KUKA KRL data list: NEW_MASTER_MESA_A.dat

&ACCESS RVP
&REL 381
&PARAM EDITMASK = *
&PARAM TEMPLATE = C:\KRC\Roboter\Template\vorgabe
&PARAM DISKPATH = KRC:\R1\Program\Solda\MASTER_125
DEFDAT  NEW_MASTER_MESA_A
;FOLD EXTERNAL DECLARATIONS;%{PE}%MKUKATPBASIS,%CEXT,%VCOMMON,%P
;FOLD BASISTECH EXT;%{PE}%MKUKATPBASIS,%CEXT,%VEXT,%P
EXT  BAS (BAS_COMMAND  :IN,REAL  :IN )
DECL INT SUCCESS
;ENDFOLD (BASISTECH EXT)
;FOLD USER EXT;%{E}%MKUKATPUSER,%CEXT,%VEXT,%P
;Make your modifications here

;ENDFOLD (USER EXT)
;ENDFOLD (EXTERNAL DECLARATIONS)
DECL ATBg_Start_T AS_WDAT1={JobModeId 1306102413,ParamSetId -1047099609,StartTime 0.0,PreFlowTime 0.0,Channel1 0.0,Channel2 2.00000,Channel3 0.0,Channel4 0.0,Channel5 0.0,Channel6 0.0,Channel7 0.0,Channel8 0.0,PurgeTime 0.0}
DECL ATBg_Weld_T AW_WDAT1={JobModeId -187662529,ParamSetId -430485013,Velocity 0.00830000,Channel1 30.0000,Channel2 1.00000,Channel3 0.0,Channel4 0.0,Channel5 0.0,Channel6 0.0,Channel7 0.0,Channel8 0.0}
DECL WTCg_WeaveDefinition_T WV_WDAT1={Pattern #None,Length 4.00000,Amplitude 2.00000,Angle 0.0}
DECL FDAT FP1={TOOL_NO 1,BASE_NO 0,IPO_FRAME #BASE,POINT2[] " ",TQ_STATE FALSE}
DECL PDAT PPDAT1={ACC 100.000,APO_DIST 100.000,APO_MODE #CPTP,GEAR_JERK 50.0000}
DECL E6POS XP1={X 1496.76196,Y 582.870911,Z 1275.91040,A 159.098511,B 49.1786919,C -124.034058,S 0,T 43,E1 180.001038,E2 179.999084,E3 180.004181,E4 0.0,E5 0.0,E6 0.0}
DECL MODULEPARAM_T LAST_TP_PARAMS={PARAMS[] "Kuka.MoveDataPtpName=PDAT60; Kuka.VelocityPtp=100; Kuka.PointName=P78; Kuka.BlendingEnabled=False; Kuka.FrameData.tq_state=False; Kuka.FrameData.base_no=0; Kuka.FrameData.tool_no=1; Kuka.FrameData.ipo_frame=#BASE; Kuka.MovementDataPdat.apo_mode=#CPTP; Kuka.MovementDataPdat.apo_dist=100; Kuka.MovementData.acc=100; Kuka.MovementData.gear_jerk=50; ArcTech.WdatVarName=WDAT39; Kuka.MoveDataName=CPDAT51; Kuka.VelocityPath=0.3; Kuka.MovementData.apo_fac=50; Kuka.MovementData.apo_dist=100; Kuka.MovementData.axis_acc=100; Kuka.MovementData.axis_vel=100; Kuka.MovementData.circ_typ=#BASE; Kuka.MovementData.exax_ign=0; Kuka.MovementData.jerk_fac=50; Kuka.MovementData.ori_typ=#VAR; Kuka.FrameData.point2=                                                                                                                                                                                                "}
DECL ATBg_Crater_T AC_WDAT2={JobModeId -187662529,ParamSetId -1375177600,CraterTime 0.100000,PostflowTime 0.100000,Channel1 30.0000,Channel2 1.00000,Channel3 0.0,Channel4 0.0,Channel5 0.0,Channel6 0.0,Channel7 0.0,Channel8 0.0,BurnBackTime 0.0}
DECL FDAT FP2={TOOL_NO 1,BASE_NO 0,IPO_FRAME #BASE,POINT2[] " ",TQ_STATE FALSE}
DECL LDAT LCPDAT1={ACC 100.000,APO_DIST 100.000,APO_FAC 50.0000,AXIS_VEL 100.000,AXIS_ACC 100.000,ORI_TYP #VAR,CIRC_TYP #BASE,JERK_FAC 50.0000,GEAR_JERK 50.0000,EXAX_IGN 0}
DECL E6POS XP2={X 1500.47852,Y 573.313171,Z 1274.83447,A 158.879135,B 49.0362473,C -123.840370,S 0,T 43,E1 180.001038,E2 179.999084,E3 180.004181,E4 0.0,E5 0.0,E6 0.0}
DECL BASIS_SUGG_T LAST_BASIS={POINT1[] "P185                    ",POINT2[] "P185                    ",CP_PARAMS[] "CPDAT0                  ",PTP_PARAMS[] "PDAT137                 ",CONT[] "C_DIS                   ",CP_VEL[] "2.0                     ",PTP_VEL[] "100                     ",SYNC_PARAMS[] "SYNCDAT                 ",SPL_NAME[] "S0                      ",A_PARAMS[] "ADAT0                   "}
DECL E6POS XP3={X 1482.70276,Y 566.674377,Z 1310.22266,A 157.428940,B 50.3861160,C -125.741325,S 0,T 43,E1 180.001038,E2 179.999084,E3 180.004181,E4 0.0,E5 0.0,E6 0.0}
DECL FDAT FP3={TOOL_NO 1,BASE_NO 0,IPO_FRAME #BASE,POINT2[] " ",TQ_STATE FALSE}
DECL PDAT PPDAT2={VEL 100.000,ACC 100.000,APO_DIST 100.000,GEAR_JERK 50.0000,EXAX_IGN 3}
DECL E6POS XP4={X 1482.70276,Y 566.674377,Z 1310.22266,A 157.428940,B 50.3861160,C -125.741325,S 0,T 43,E1 180.001038,E2 179.999084,E3 180.004181,E4 0.0,E5 0.0,E6 0.0}
DECL FDAT FP4={TOOL_NO 1,BASE_NO 0,IPO_FRAME #BASE,POINT2[] " ",TQ_STATE FALSE}
DECL PDAT PPDAT3={VEL 100.000,ACC 100.000,APO_DIST 100.000,GEAR_JERK 50.0000,EXAX_IGN 3}
DECL ATBg_Start_T AS_WDAT3={JobModeId 1306102413,ParamSetId -1047099609,StartTime 0.0,PreFlowTime 0.0,Channel1 0.0,Channel2 2.00000,Channel3 0.0,Channel4 0.0,Channel5 0.0,Channel6 0.0,Channel7 0.0,Channel8 0.0,PurgeTime 0.0}
DECL ATBg_Weld_T AW_WDAT3={JobModeId -187662529,ParamSetId -430485013,Velocity 0.00830000,Channel1 30.0000,Channel2 1.00000,Channel3 0.0,Channel4 0.0,Channel5 0.0,Channel6 0.0,Channel7 0.0,Channel8 0.0}
DECL WTCg_WeaveDefinition_T WV_WDAT3={Pattern #None,Length 4.00000,Amplitude 2.00000,Angle 0.0}
DECL FDAT FP5={TOOL_NO 1,BASE_NO 0,IPO_FRAME #BASE,POINT2[] " ",TQ_STATE FALSE}
DECL PDAT PPDAT4={ACC 100.000,APO_DIST 100.000,APO_MODE #CPTP,GEAR_JERK 50.0000}
DECL E6POS XP5={X 1466.55981,Y 697.098694,Z 1383.56360,A -77.2453308,B 24.5325470,C -35.8039818,S 0,T 11,E1 180.001022,E2 179.999100,E3 180.004028,E4 0.0,E5 0.0,E6 0.0}
DECL ATBg_Crater_T AC_WDAT4={JobModeId -187662529,ParamSetId -1375177600,CraterTime 0.100000,PostflowTime 0.100000,Channel1 30.0000,Channel2 1.00000,Channel3 0.0,Channel4 0.0,Channel5 0.0,Channel6 0.0,Channel7 0.0,Channel8 0.0,BurnBackTime 0.0}
DECL FDAT FP6={TOOL_NO 1,BASE_NO 0,IPO_FRAME #BASE,POINT2[] " ",TQ_STATE FALSE}
DECL LDAT LCPDAT2={ACC 100.000,APO_DIST 100.000,APO_FAC 50.0000,AXIS_VEL 100.000,AXIS_ACC 100.000,ORI_TYP #VAR,CIRC_TYP #BASE,JERK_FAC 50.0000,GEAR_JERK 50.0000,EXAX_IGN 0}
DECL E6POS XP6={X 1461.39319,Y 705.430176,Z 1377.38342,A -77.4356918,B 24.1875134,C -37.1046600,S 2,T 11,E1 180.001022,E2 179.999100,E3 180.004028,E4 0.0,E5 0.0,E6 0.0}
DECL LDAT LCPDAT3={ACC 100.000,APO_DIST 100.000,APO_FAC 50.0000,AXIS_VEL 100.000,AXIS_ACC 100.000,ORI_TYP #VAR,CIRC_TYP #BASE,JERK_FAC 50.0000,GEAR_JERK 50.0000,EXAX_IGN 0}
DECL LDAT LCPDAT4={ACC 100.000,APO_DIST 100.000,APO_FAC 50.0000,AXIS_VEL 100.000,AXIS_ACC 100.000,ORI_TYP #VAR,CIRC_TYP #BASE,JERK_FAC 50.0000,GEAR_JERK 50.0000,EXAX_IGN 0}
DECL PDAT PPDAT5={ACC 100.000,APO_DIST 100.000,APO_MODE #CPTP,GEAR_JERK 50.0000}
DECL ATBg_Start_T AS_WDAT5={JobModeId 1306102413,ParamSetId -1047099609,StartTime 0.0,PreFlowTime 0.0,Channel1 0.0,Channel2 2.00000,Channel3 0.0,Channel4 0.0,Channel5 0.0,Channel6 0.0,Channel7 0.0,Channel8 0.0,PurgeTime 0.0}
DECL ATBg_Weld_T AW_WDAT5={JobModeId -187662529,ParamSetId -430485013,Velocity 0.00830000,Channel1 30.0000,Channel2 1.00000,Channel3 0.0,Channel4 0.0,Channel5 0.0,Channel6 0.0,Channel7 0.0,Channel8 0.0}
DECL WTCg_WeaveDefinition_T WV_WDAT5={Pattern #None,Length 4.00000,Amplitude 2.00000,Angle 0.0}
DECL FDAT FP7={TOOL_NO 1,BASE_NO 0,IPO_FRAME #BASE,POINT2[] " ",TQ_STATE FALSE}
DECL PDAT PPDAT6={ACC 100.000,APO_DIST 100.000,APO_MODE #CPTP,GEAR_JERK 50.0000}
DECL E6POS XP7={X 1484.82764,Y 693.075134,Z 1499.31616,A -23.4080772,B -53.4302559,C -46.9197922,S 2,T 43,E1 180.001022,E2 179.999100,E3 180.004028,E4 0.0,E5 0.0,E6 0.0}
DECL ATBg_Crater_T AC_WDAT6={JobModeId -187662529,ParamSetId -1375177600,CraterTime 0.100000,PostflowTime 0.100000,Channel1 30.0000,Channel2 1.00000,Channel3 0.0,Channel4 0.0,Channel5 0.0,Channel6 0.0,Channel7 0.0,Channel8 0.0,BurnBackTime 0.0}
DECL FDAT FP8={TOOL_NO 1,BASE_NO 0,IPO_FRAME #BASE,POINT2[] " ",TQ_STATE FALSE}
DECL LDAT LCPDAT5={ACC 100.000,APO_DIST 100.000,APO_FAC 50.0000,AXIS_VEL 100.000,AXIS_ACC 100.000,ORI_TYP #VAR,CIRC_TYP #BASE,JERK_FAC 50.0000,GEAR_JERK 50.0000,EXAX_IGN 0}
DECL E6POS XP8={X 1489.87585,Y 680.574158,Z 1497.46960,A -29.8228798,B -49.4180946,C -42.0220261,S 2,T 43,E1 180.001022,E2 179.999100,E3 180.004028,E4 0.0,E5 0.0,E6 0.0}
DECL E6POS XP9={X 1436.40173,Y 655.308228,Z 1566.53308,A -32.0819,B -50.6817131,C -39.0761185,S 2,T 43,E1 180.000992,E2 179.999115,E3 180.003891,E4 0.0,E5 0.0,E6 0.0}
DECL FDAT FP9={TOOL_NO 1,BASE_NO 0,IPO_FRAME #BASE,POINT2[] " ",TQ_STATE FALSE}
DECL PDAT PPDAT7={VEL 100.000,ACC 100.000,APO_DIST 100.000,GEAR_JERK 50.0000,EXAX_IGN 3}
DECL E6POS XP10={X 1436.40173,Y 655.308228,Z 1566.53308,A -32.0819,B -50.6817131,C -39.0761185,S 2,T 43,E1 180.000992,E2 179.999115,E3 180.003891,E4 0.0,E5 0.0,E6 0.0}
DECL FDAT FP10={TOOL_NO 1,BASE_NO 0,IPO_FRAME #BASE,POINT2[] " ",TQ_STATE FALSE}
DECL PDAT PPDAT8={VEL 100.000,ACC 100.000,APO_DIST 100.000,GEAR_JERK 50.0000,EXAX_IGN 3}
DECL E6POS XP11={X 963.610474,Y 468.452576,Z 2013.77759,A -55.0418549,B -77.1242065,C -9.45068359,S 2,T 43,E1 180.000992,E2 179.999115,E3 180.003891,E4 0.0,E5 0.0,E6 0.0}
DECL FDAT FP11={TOOL_NO 1,BASE_NO 0,IPO_FRAME #BASE,POINT2[] " ",TQ_STATE FALSE}
DECL PDAT PPDAT9={VEL 100.000,ACC 100.000,APO_DIST 100.000,GEAR_JERK 50.0000,EXAX_IGN 3}
DECL E6POS XP12={X 1030.98926,Y 213.392715,Z 1949.10840,A -48.0140724,B -75.1600342,C -31.3416386,S 2,T 43,E1 180.000992,E2 179.999115,E3 180.003891,E4 0.0,E5 0.0,E6 0.0}
DECL FDAT FP12={TOOL_NO 1,BASE_NO 0,IPO_FRAME #BASE,POINT2[] " ",TQ_STATE FALSE}
DECL PDAT PPDAT10={VEL 100.000,ACC 100.000,APO_DIST 100.000,GEAR_JERK 50.0000,EXAX_IGN 3}
DECL E6POS XP13={X 1582.72571,Y 214.898727,Z 1484.79297,A -17.8722897,B -60.1868629,C -67.3960724,S 2,T 43,E1 180.000992,E2 179.999115,E3 180.003891,E4 0.0,E5 0.0,E6 0.0}
DECL FDAT FP13={TOOL_NO 1,BASE_NO 0,IPO_FRAME #BASE,POINT2[] " ",TQ_STATE FALSE}
DECL PDAT PPDAT11={VEL 100.000,ACC 100.000,APO_DIST 100.000,GEAR_JERK 50.0000,EXAX_IGN 3}
DECL ATBg_Start_T AS_WDAT7={JobModeId 1306102413,ParamSetId -1047099609,StartTime 0.0,PreFlowTime 0.0,Channel1 0.0,Channel2 2.00000,Channel3 0.0,Channel4 0.0,Channel5 0.0,Channel6 0.0,Channel7 0.0,Channel8 0.0,PurgeTime 0.0}
DECL ATBg_Weld_T AW_WDAT7={JobModeId -187662529,ParamSetId -430485013,Velocity 0.00830000,Channel1 30.0000,Channel2 1.00000,Channel3 0.0,Channel4 0.0,Channel5 0.0,Channel6 0.0,Channel7 0.0,Channel8 0.0}
DECL WTCg_WeaveDefinition_T WV_WDAT7={Pattern #None,Length 4.00000,Amplitude 2.00000,Angle 0.0}
DECL FDAT FP14={TOOL_NO 1,BASE_NO 0,IPO_FRAME #BASE,POINT2[] " ",TQ_STATE FALSE}
DECL PDAT PPDAT12={ACC 100.000,APO_DIST 100.000,APO_MODE #CPTP,GEAR_JERK 50.0000}
DECL E6POS XP14={X 1584.62036,Y 215.140686,Z 1482.90674,A -17.8341675,B -60.1402512,C -67.4400177,S 2,T 43,E1 180.000992,E2 179.999115,E3 180.003891,E4 0.0,E5 0.0,E6 0.0}
DECL ATBg_Crater_T AC_WDAT8={JobModeId -187662529,ParamSetId -1375177600,CraterTime 0.100000,PostflowTime 0.100000,Channel1 30.0000,Channel2 1.00000,Channel3 0.0,Channel4 0.0,Channel5 0.0,Channel6 0.0,Channel7 0.0,Channel8 0.0,BurnBackTime 0.0}
DECL FDAT FP15={TOOL_NO 1,BASE_NO 0,IPO_FRAME #BASE,POINT2[] " ",TQ_STATE FALSE}
DECL LDAT LCPDAT6={ACC 100.000,APO_DIST 100.000,APO_FAC 50.0000,AXIS_VEL 100.000,AXIS_ACC 100.000,ORI_TYP #VAR,CIRC_TYP #BASE,JERK_FAC 50.0000,GEAR_JERK 50.0000,EXAX_IGN 0}
DECL E6POS XP15={X 1584.62036,Y 215.140686,Z 1482.90674,A -17.8341675,B -60.1402512,C -67.4400177,S 2,T 43,E1 180.000992,E2 179.999115,E3 180.003891,E4 0.0,E5 0.0,E6 0.0}
DECL E6POS XP16={X 1547.48352,Y 210.398209,Z 1520.88965,A -18.7159042,B -61.1769409,C -66.4285660,S 2,T 43,E1 180.000992,E2 179.999115,E3 180.003891,E4 0.0,E5 0.0,E6 0.0}
DECL FDAT FP16={TOOL_NO 1,BASE_NO 0,IPO_FRAME #BASE,POINT2[] " ",TQ_STATE FALSE}
DECL PDAT PPDAT13={VEL 100.000,ACC 100.000,APO_DIST 100.000,GEAR_JERK 50.0000,EXAX_IGN 3}
DECL E6POS XP17={X 1505.81213,Y 205.076660,Z 1574.12085,A -20.5965290,B -63.1322670,C -64.3020325,S 2,T 43,E1 180.000992,E2 179.999115,E3 180.003891,E4 0.0,E5 0.0,E6 0.0}
DECL FDAT FP17={TOOL_NO 1,BASE_NO 0,IPO_FRAME #BASE,POINT2[] " ",TQ_STATE FALSE}
DECL PDAT PPDAT14={VEL 100.000,ACC 100.000,APO_DIST 100.000,GEAR_JERK 50.0000,EXAX_IGN 3}
DECL E6POS XP18={X 1562.25806,Y 172.455948,Z 1399.03113,A -178.023010,B 72.2041321,C -95.4785080,S 2,T 43,E1 180.000992,E2 179.999115,E3 180.003891,E4 0.0,E5 0.0,E6 0.0}
DECL FDAT FP18={TOOL_NO 1,BASE_NO 0,IPO_FRAME #BASE,POINT2[] " ",TQ_STATE FALSE}
DECL PDAT PPDAT15={VEL 100.000,ACC 100.000,APO_DIST 100.000,GEAR_JERK 50.0000,EXAX_IGN 3}
DECL ATBg_Start_T AS_WDAT9={JobModeId 1306102413,ParamSetId -1047099609,StartTime 0.0,PreFlowTime 0.0,Channel1 0.0,Channel2 2.00000,Channel3 0.0,Channel4 0.0,Channel5 0.0,Channel6 0.0,Channel7 0.0,Channel8 0.0,PurgeTime 0.0}
DECL ATBg_Weld_T AW_WDAT9={JobModeId -187662529,ParamSetId -430485013,Velocity 0.00830000,Channel1 30.0000,Channel2 1.00000,Channel3 0.0,Channel4 0.0,Channel5 0.0,Channel6 0.0,Channel7 0.0,Channel8 0.0}
DECL WTCg_WeaveDefinition_T WV_WDAT9={Pattern #None,Length 4.00000,Amplitude 2.00000,Angle 0.0}
DECL FDAT FP19={TOOL_NO 1,BASE_NO 0,IPO_FRAME #BASE,POINT2[] " ",TQ_STATE FALSE}
DECL PDAT PPDAT16={ACC 100.000,APO_DIST 100.000,APO_MODE #CPTP,GEAR_JERK 50.0000}
DECL E6POS XP19={X 1594.61816,Y 176.588425,Z 1348.24695,A -177.500946,B 70.1884537,C -94.9270935,S 2,T 43,E1 180.000992,E2 179.999115,E3 180.003891,E4 0.0,E5 0.0,E6 0.0}
DECL ATBg_Crater_T AC_WDAT10={JobModeId -187662529,ParamSetId -1375177600,CraterTime 0.100000,PostflowTime 0.100000,Channel1 30.0000,Channel2 1.00000,Channel3 0.0,Channel4 0.0,Channel5 0.0,Channel6 0.0,Channel7 0.0,Channel8 0.0,BurnBackTime 0.0}
DECL FDAT FP20={TOOL_NO 1,BASE_NO 0,IPO_FRAME #BASE,POINT2[] " ",TQ_STATE FALSE}
DECL LDAT LCPDAT7={ACC 100.000,APO_DIST 100.000,APO_FAC 50.0000,AXIS_VEL 100.000,AXIS_ACC 100.000,ORI_TYP #VAR,CIRC_TYP #BASE,JERK_FAC 50.0000,GEAR_JERK 50.0000,EXAX_IGN 0}
DECL E6POS XP20={X 1594.61816,Y 176.588425,Z 1348.24695,A -177.500946,B 70.1884537,C -94.9270935,S 2,T 43,E1 180.000992,E2 179.999115,E3 180.003891,E4 0.0,E5 0.0,E6 0.0}
DECL E6POS XP21={X 1562.25806,Y 172.455933,Z 1399.03113,A -178.023010,B 72.2041321,C -95.4785080,S 2,T 43,E1 180.000992,E2 179.999115,E3 180.003891,E4 0.0,E5 0.0,E6 0.0}
DECL FDAT FP21={TOOL_NO 1,BASE_NO 0,IPO_FRAME #BASE,POINT2[] " ",TQ_STATE FALSE}
DECL PDAT PPDAT17={VEL 100.000,ACC 100.000,APO_DIST 100.000,GEAR_JERK 50.0000,EXAX_IGN 3}
DECL E6POS XP22={X 1528.15576,Y 167.507034,Z 1565.51379,A 28.2313652,B 85.1708,C 110.647263,S 2,T 43,E1 180.000992,E2 179.999115,E3 180.003891,E4 0.0,E5 0.0,E6 0.0}
DECL FDAT FP22={TOOL_NO 1,BASE_NO 0,IPO_FRAME #BASE,POINT2[] " ",TQ_STATE FALSE}
DECL PDAT PPDAT18={VEL 100.000,ACC 100.000,APO_DIST 100.000,GEAR_JERK 50.0000,EXAX_IGN 3}
DECL E6POS XP23={X 1502.60278,Y -324.416138,Z 1572.55701,A -74.3732529,B 79.7488556,C 26.2741585,S 2,T 10,E1 180.000992,E2 179.999115,E3 180.003891,E4 0.0,E5 0.0,E6 0.0}
DECL FDAT FP23={TOOL_NO 1,BASE_NO 0,IPO_FRAME #BASE,POINT2[] " ",TQ_STATE FALSE}
DECL PDAT PPDAT19={VEL 100.000,ACC 100.000,APO_DIST 100.000,GEAR_JERK 50.0000,EXAX_IGN 3}
DECL ATBg_Start_T AS_WDAT11={JobModeId 1306102413,ParamSetId -1047099609,StartTime 0.0,PreFlowTime 0.0,Channel1 0.0,Channel2 2.00000,Channel3 0.0,Channel4 0.0,Channel5 0.0,Channel6 0.0,Channel7 0.0,Channel8 0.0,PurgeTime 0.0}
DECL ATBg_Weld_T AW_WDAT11={JobModeId -187662529,ParamSetId -430485013,Velocity 0.00830000,Channel1 30.0000,Channel2 1.00000,Channel3 0.0,Channel4 0.0,Channel5 0.0,Channel6 0.0,Channel7 0.0,Channel8 0.0}
DECL WTCg_WeaveDefinition_T WV_WDAT11={Pattern #None,Length 4.00000,Amplitude 2.00000,Angle 0.0}
DECL FDAT FP24={TOOL_NO 1,BASE_NO 0,IPO_FRAME #BASE,POINT2[] " ",TQ_STATE FALSE}
DECL PDAT PPDAT20={ACC 100.000,APO_DIST 100.000,APO_MODE #CPTP,GEAR_JERK 50.0000}
DECL E6POS XP24={X 1574.90735,Y -337.206,Z 1350.69495,A -165.207779,B 67.7758102,C -66.7983551,S 2,T 10,E1 180.000992,E2 179.999115,E3 180.003891,E4 0.0,E5 0.0,E6 0.0}
DECL ATBg_Crater_T AC_WDAT12={JobModeId -187662529,ParamSetId -1375177600,CraterTime 0.100000,PostflowTime 0.100000,Channel1 30.0000,Channel2 1.00000,Channel3 0.0,Channel4 0.0,Channel5 0.0,Channel6 0.0,Channel7 0.0,Channel8 0.0,BurnBackTime 0.0}
DECL FDAT FP25={TOOL_NO 1,BASE_NO 0,IPO_FRAME #BASE,POINT2[] " ",TQ_STATE FALSE}
DECL LDAT LCPDAT8={ACC 100.000,APO_DIST 100.000,APO_FAC 50.0000,AXIS_VEL 100.000,AXIS_ACC 100.000,ORI_TYP #VAR,CIRC_TYP #BASE,JERK_FAC 50.0000,GEAR_JERK 50.0000,EXAX_IGN 0}
DECL E6POS XP25={X 1574.90735,Y -337.206,Z 1350.69495,A -165.207779,B 67.7758102,C -66.7983551,S 2,T 10,E1 180.000992,E2 179.999115,E3 180.003891,E4 0.0,E5 0.0,E6 0.0}
DECL E6POS XP26={X 1522.26257,Y -327.427399,Z 1432.21021,A -161.269516,B 70.6730652,C -62.5877876,S 2,T 10,E1 180.000992,E2 179.999115,E3 180.003891,E4 0.0,E5 0.0,E6 0.0}
DECL FDAT FP26={TOOL_NO 1,BASE_NO 0,IPO_FRAME #BASE,POINT2[] " ",TQ_STATE FALSE}
DECL PDAT PPDAT21={VEL 100.000,ACC 100.000,APO_DIST 100.000,GEAR_JERK 50.0000,EXAX_IGN 3}
DECL E6POS XP27={X 1491.06848,Y -228.728851,Z 1583.72083,A 11.7713518,B -64.7742691,C -109.904411,S 2,T 10,E1 180.000992,E2 179.999115,E3 180.003891,E4 0.0,E5 0.0,E6 0.0}
DECL FDAT FP27={TOOL_NO 1,BASE_NO 0,IPO_FRAME #BASE,POINT2[] " ",TQ_STATE FALSE}
DECL PDAT PPDAT22={VEL 100.000,ACC 100.000,APO_DIST 100.000,GEAR_JERK 50.0000,EXAX_IGN 3}
DECL ATBg_Start_T AS_WDAT13={JobModeId 1306102413,ParamSetId -1047099609,StartTime 0.0,PreFlowTime 0.0,Channel1 0.0,Channel2 2.00000,Channel3 0.0,Channel4 0.0,Channel5 0.0,Channel6 0.0,Channel7 0.0,Channel8 0.0,PurgeTime 0.0}
DECL ATBg_Weld_T AW_WDAT13={JobModeId -187662529,ParamSetId -430485013,Velocity 0.00830000,Channel1 30.0000,Channel2 1.00000,Channel3 0.0,Channel4 0.0,Channel5 0.0,Channel6 0.0,Channel7 0.0,Channel8 0.0}
DECL WTCg_WeaveDefinition_T WV_WDAT13={Pattern #None,Length 4.00000,Amplitude 2.00000,Angle 0.0}
DECL FDAT FP28={TOOL_NO 1,BASE_NO 0,IPO_FRAME #BASE,POINT2[] " ",TQ_STATE FALSE}
DECL PDAT PPDAT23={ACC 100.000,APO_DIST 100.000,APO_MODE #CPTP,GEAR_JERK 50.0000}
DECL E6POS XP28={X 1572.85193,Y -243.939880,Z 1478.24158,A 8.99041462,B -61.0612869,C -106.788139,S 2,T 10,E1 180.000992,E2 179.999115,E3 180.003891,E4 0.0,E5 0.0,E6 0.0}
DECL ATBg_Crater_T AC_WDAT14={JobModeId -187662529,ParamSetId -1375177600,CraterTime 0.100000,PostflowTime 0.100000,Channel1 30.0000,Channel2 1.00000,Channel3 0.0,Channel4 0.0,Channel5 0.0,Channel6 0.0,Channel7 0.0,Channel8 0.0,BurnBackTime 0.0}
DECL FDAT FP29={TOOL_NO 1,BASE_NO 0,IPO_FRAME #BASE,POINT2[] " ",TQ_STATE FALSE}
DECL LDAT LCPDAT9={ACC 100.000,APO_DIST 100.000,APO_FAC 50.0000,AXIS_VEL 100.000,AXIS_ACC 100.000,ORI_TYP #VAR,CIRC_TYP #BASE,JERK_FAC 50.0000,GEAR_JERK 50.0000,EXAX_IGN 0}
DECL E6POS XP29={X 1572.85193,Y -243.939880,Z 1478.24158,A 8.99041462,B -61.0612869,C -106.788139,S 2,T 10,E1 180.000992,E2 179.999115,E3 180.003891,E4 0.0,E5 0.0,E6 0.0}
DECL E6POS XP30={X 1435.31335,Y -218.392578,Z 1621.85400,A 12.7399940,B -65.8434830,C -110.975647,S 2,T 10,E1 180.000992,E2 179.999115,E3 180.003891,E4 0.0,E5 0.0,E6 0.0}
DECL FDAT FP30={TOOL_NO 1,BASE_NO 0,IPO_FRAME #BASE,POINT2[] " ",TQ_STATE FALSE}
DECL PDAT PPDAT24={VEL 100.000,ACC 100.000,APO_DIST 100.000,GEAR_JERK 50.0000,EXAX_IGN 3}
DECL E6POS XP31={X 1211.71753,Y -176.207092,Z 1775.64709,A 10.2153435,B -62.4659920,C -107.999146,S 2,T 10,E1 180.000992,E2 179.999115,E3 180.003891,E4 0.0,E5 0.0,E6 0.0}
DECL FDAT FP31={TOOL_NO 1,BASE_NO 0,IPO_FRAME #BASE,POINT2[] " ",TQ_STATE FALSE}
DECL PDAT PPDAT25={VEL 100.000,ACC 100.000,APO_DIST 100.000,GEAR_JERK 50.0000,EXAX_IGN 3}
DECL E6POS XP32={X 1115.09851,Y -492.561127,Z 1780.23438,A 33.0263557,B -54.0004311,C -144.370392,S 2,T 10,E1 180.000992,E2 179.999115,E3 180.003891,E4 0.0,E5 0.0,E6 0.0}
DECL FDAT FP32={TOOL_NO 1,BASE_NO 0,IPO_FRAME #BASE,POINT2[] " ",TQ_STATE FALSE}
DECL PDAT PPDAT26={VEL 100.000,ACC 100.000,APO_DIST 100.000,GEAR_JERK 50.0000,EXAX_IGN 3}
DECL ATBg_Start_T AS_WDAT15={JobModeId 1306102413,ParamSetId -1047099609,StartTime 0.0,PreFlowTime 0.0,Channel1 0.0,Channel2 2.00000,Channel3 0.0,Channel4 0.0,Channel5 0.0,Channel6 0.0,Channel7 0.0,Channel8 0.0,PurgeTime 0.0}
DECL ATBg_Weld_T AW_WDAT15={JobModeId -187662529,ParamSetId -430485013,Velocity 0.00830000,Channel1 30.0000,Channel2 1.00000,Channel3 0.0,Channel4 0.0,Channel5 0.0,Channel6 0.0,Channel7 0.0,Channel8 0.0}
DECL WTCg_WeaveDefinition_T WV_WDAT15={Pattern #None,Length 4.00000,Amplitude 2.00000,Angle 0.0}
DECL FDAT FP33={TOOL_NO 1,BASE_NO 0,IPO_FRAME #BASE,POINT2[] " ",TQ_STATE FALSE}
DECL PDAT PPDAT27={ACC 100.000,APO_DIST 100.000,APO_MODE #CPTP,GEAR_JERK 50.0000}
DECL E6POS XP33={X 1497.54565,Y -521.613,Z 1444.21875,A 57.3688469,B 47.0705,C 163.948288,S 6,T 58,E1 180.000992,E2 179.999115,E3 180.003891,E4 0.0,E5 0.0,E6 0.0}
DECL ATBg_Crater_T AC_WDAT16={JobModeId -187662529,ParamSetId -1375177600,CraterTime 0.100000,PostflowTime 0.100000,Channel1 30.0000,Channel2 1.00000,Channel3 0.0,Channel4 0.0,Channel5 0.0,Channel6 0.0,Channel7 0.0,Channel8 0.0,BurnBackTime 0.0}
DECL FDAT FP34={TOOL_NO 1,BASE_NO 0,IPO_FRAME #BASE,POINT2[] " ",TQ_STATE FALSE}
DECL LDAT LCPDAT10={ACC 100.000,APO_DIST 100.000,APO_FAC 50.0000,AXIS_VEL 100.000,AXIS_ACC 100.000,ORI_TYP #VAR,CIRC_TYP #BASE,JERK_FAC 50.0000,GEAR_JERK 50.0000,EXAX_IGN 0}
DECL E6POS XP34={X 1497.54565,Y -521.613,Z 1444.21875,A 57.3688469,B 47.0705,C 163.948288,S 6,T 58,E1 180.000992,E2 179.999115,E3 180.003891,E4 0.0,E5 0.0,E6 0.0}
DECL ATBg_Start_T AS_WDAT17={JobModeId 1306102413,ParamSetId -1047099609,StartTime 0.0,PreFlowTime 0.0,Channel1 0.0,Channel2 2.00000,Channel3 0.0,Channel4 0.0,Channel5 0.0,Channel6 0.0,Channel7 0.0,Channel8 0.0,PurgeTime 0.0}
DECL ATBg_Weld_T AW_WDAT17={JobModeId -187662529,ParamSetId -430485013,Velocity 0.00830000,Channel1 30.0000,Channel2 1.00000,Channel3 0.0,Channel4 0.0,Channel5 0.0,Channel6 0.0,Channel7 0.0,Channel8 0.0}
DECL WTCg_WeaveDefinition_T WV_WDAT17={Pattern #None,Length 4.00000,Amplitude 2.00000,Angle 0.0}
DECL FDAT FP35={TOOL_NO 1,BASE_NO 0,IPO_FRAME #BASE,POINT2[] " ",TQ_STATE FALSE}
DECL PDAT PPDAT28={ACC 100.000,APO_DIST 100.000,APO_MODE #CPTP,GEAR_JERK 50.0000}
DECL E6POS XP35={X 1490.85339,Y -544.309875,Z 1445.73792,A 56.1921425,B 47.0849609,C 163.538742,S 6,T 58,E1 180.000992,E2 179.999115,E3 180.003891,E4 0.0,E5 0.0,E6 0.0}
DECL ATBg_Crater_T AC_WDAT18={JobModeId -187662529,ParamSetId -1375177600,CraterTime 0.100000,PostflowTime 0.100000,Channel1 30.0000,Channel2 1.00000,Channel3 0.0,Channel4 0.0,Channel5 0.0,Channel6 0.0,Channel7 0.0,Channel8 0.0,BurnBackTime 0.0}
DECL FDAT FP36={TOOL_NO 1,BASE_NO 0,IPO_FRAME #BASE,POINT2[] " ",TQ_STATE FALSE}
DECL LDAT LCPDAT11={ACC 100.000,APO_DIST 100.000,APO_FAC 50.0000,AXIS_VEL 100.000,AXIS_ACC 100.000,ORI_TYP #VAR,CIRC_TYP #BASE,JERK_FAC 50.0000,GEAR_JERK 50.0000,EXAX_IGN 0}
DECL E6POS XP36={X 1490.85339,Y -544.309875,Z 1445.73792,A 56.1921425,B 47.0849609,C 163.538742,S 6,T 58,E1 180.000992,E2 179.999115,E3 180.003891,E4 0.0,E5 0.0,E6 0.0}
DECL ATBg_Start_T AS_WDAT19={JobModeId 1306102413,ParamSetId -1047099609,StartTime 0.0,PreFlowTime 0.0,Channel1 0.0,Channel2 2.00000,Channel3 0.0,Channel4 0.0,Channel5 0.0,Channel6 0.0,Channel7 0.0,Channel8 0.0,PurgeTime 0.0}
DECL ATBg_Weld_T AW_WDAT19={JobModeId -187662529,ParamSetId -430485013,Velocity 0.00830000,Channel1 30.0000,Channel2 1.00000,Channel3 0.0,Channel4 0.0,Channel5 0.0,Channel6 0.0,Channel7 0.0,Channel8 0.0}
DECL WTCg_WeaveDefinition_T WV_WDAT19={Pattern #None,Length 4.00000,Amplitude 2.00000,Angle 0.0}
DECL FDAT FP37={TOOL_NO 1,BASE_NO 0,IPO_FRAME #BASE,POINT2[] " ",TQ_STATE FALSE}
DECL PDAT PPDAT29={ACC 100.000,APO_DIST 100.000,APO_MODE #CPTP,GEAR_JERK 50.0000}
DECL E6POS XP37={X 1451.87244,Y -698.568726,Z 1532.68176,A -109.570,B -5.58304501,C 1.80761051,S 2,T 42,E1 180.000992,E2 179.999115,E3 180.003891,E4 0.0,E5 0.0,E6 0.0}
DECL ATBg_Crater_T AC_WDAT20={JobModeId -187662529,ParamSetId -1375177600,CraterTime 0.100000,PostflowTime 0.100000,Channel1 30.0000,Channel2 1.00000,Channel3 0.0,Channel4 0.0,Channel5 0.0,Channel6 0.0,Channel7 0.0,Channel8 0.0,BurnBackTime 0.0}
DECL FDAT FP38={TOOL_NO 1,BASE_NO 0,IPO_FRAME #BASE,POINT2[] " ",TQ_STATE FALSE}
DECL LDAT LCPDAT12={ACC 100.000,APO_DIST 100.000,APO_FAC 50.0000,AXIS_VEL 100.000,AXIS_ACC 100.000,ORI_TYP #VAR,CIRC_TYP #BASE,JERK_FAC 50.0000,GEAR_JERK 50.0000,EXAX_IGN 0}
DECL E6POS XP38={X 1451.87244,Y -698.568726,Z 1532.68176,A -109.570,B -5.58304501,C 1.80761051,S 2,T 42,E1 180.000992,E2 179.999115,E3 180.003891,E4 0.0,E5 0.0,E6 0.0}
DECL ATBg_Start_T AS_WDAT21={JobModeId 1306102413,ParamSetId -1047099609,StartTime 0.0,PreFlowTime 0.0,Channel1 0.0,Channel2 2.00000,Channel3 0.0,Channel4 0.0,Channel5 0.0,Channel6 0.0,Channel7 0.0,Channel8 0.0,PurgeTime 0.0}
DECL ATBg_Weld_T AW_WDAT21={JobModeId -187662529,ParamSetId -430485013,Velocity 0.00830000,Channel1 30.0000,Channel2 1.00000,Channel3 0.0,Channel4 0.0,Channel5 0.0,Channel6 0.0,Channel7 0.0,Channel8 0.0}
DECL WTCg_WeaveDefinition_T WV_WDAT21={Pattern #None,Length 4.00000,Amplitude 2.00000,Angle 0.0}
DECL FDAT FP39={TOOL_NO 1,BASE_NO 0,IPO_FRAME #BASE,POINT2[] " ",TQ_STATE FALSE}
DECL PDAT PPDAT30={ACC 100.000,APO_DIST 100.000,APO_MODE #CPTP,GEAR_JERK 50.0000}
DECL E6POS XP39={X 1465.31274,Y -658.103333,Z 1529.15979,A -108.004921,B -5.55257273,C 1.30878568,S 2,T 42,E1 180.000992,E2 179.999115,E3 180.003891,E4 0.0,E5 0.0,E6 0.0}
DECL ATBg_Crater_T AC_WDAT22={JobModeId -187662529,ParamSetId -1375177600,CraterTime 0.100000,PostflowTime 0.100000,Channel1 30.0000,Channel2 1.00000,Channel3 0.0,Channel4 0.0,Channel5 0.0,Channel6 0.0,Channel7 0.0,Channel8 0.0,BurnBackTime 0.0}
DECL FDAT FP40={TOOL_NO 1,BASE_NO 0,IPO_FRAME #BASE,POINT2[] " ",TQ_STATE FALSE}
DECL LDAT LCPDAT13={ACC 100.000,APO_DIST 100.000,APO_FAC 50.0000,AXIS_VEL 100.000,AXIS_ACC 100.000,ORI_TYP #VAR,CIRC_TYP #BASE,JERK_FAC 50.0000,GEAR_JERK 50.0000,EXAX_IGN 0}
DECL E6POS XP40={X 1465.31274,Y -658.103333,Z 1529.15979,A -108.004921,B -5.55257273,C 1.30878568,S 2,T 42,E1 180.000992,E2 179.999115,E3 180.003891,E4 0.0,E5 0.0,E6 0.0}
DECL E6POS XP41={X 1407.73132,Y -635.373413,Z 1607.95020,A -108.317863,B -5.73952579,C 4.48886776,S 2,T 42,E1 180.000992,E2 179.999115,E3 180.003891,E4 0.0,E5 0.0,E6 0.0}
DECL FDAT FP41={TOOL_NO 1,BASE_NO 0,IPO_FRAME #BASE,POINT2[] " ",TQ_STATE FALSE}
DECL PDAT PPDAT31={VEL 100.000,ACC 100.000,APO_DIST 100.000,GEAR_JERK 50.0000,EXAX_IGN 3}
DECL E6POS XP42={X 1421.12781,Y -644.572815,Z 1538.56335,A -91.9589157,B 50.3912086,C 18.5021782,S 2,T 42,E1 180.000992,E2 179.999115,E3 180.003891,E4 0.0,E5 0.0,E6 0.0}
DECL FDAT FP42={TOOL_NO 1,BASE_NO 0,IPO_FRAME #BASE,POINT2[] " ",TQ_STATE FALSE}
DECL PDAT PPDAT32={VEL 100.000,ACC 100.000,APO_DIST 100.000,GEAR_JERK 50.0000,EXAX_IGN 3}
DECL ATBg_Start_T AS_WDAT23={JobModeId 1306102413,ParamSetId -1047099609,StartTime 0.0,PreFlowTime 0.0,Channel1 0.0,Channel2 2.00000,Channel3 0.0,Channel4 0.0,Channel5 0.0,Channel6 0.0,Channel7 0.0,Channel8 0.0,PurgeTime 0.0}
DECL ATBg_Weld_T AW_WDAT23={JobModeId -187662529,ParamSetId -430485013,Velocity 0.00830000,Channel1 30.0000,Channel2 1.00000,Channel3 0.0,Channel4 0.0,Channel5 0.0,Channel6 0.0,Channel7 0.0,Channel8 0.0}
DECL WTCg_WeaveDefinition_T WV_WDAT23={Pattern #None,Length 4.00000,Amplitude 2.00000,Angle 0.0}
DECL FDAT FP43={TOOL_NO 1,BASE_NO 0,IPO_FRAME #BASE,POINT2[] " ",TQ_STATE FALSE}
DECL PDAT PPDAT33={ACC 100.000,APO_DIST 100.000,APO_MODE #CPTP,GEAR_JERK 50.0000}
DECL E6POS XP43={X 1502.02258,Y -578.292908,Z 1485.39441,A 30.5960255,B -59.1033821,C -140.023438,S 2,T 34,E1 180.000992,E2 179.999115,E3 180.003891,E4 0.0,E5 0.0,E6 0.0}
DECL ATBg_Crater_T AC_WDAT24={JobModeId -187662529,ParamSetId -1375177600,CraterTime 0.100000,PostflowTime 0.100000,Channel1 30.0000,Channel2 1.00000,Channel3 0.0,Channel4 0.0,Channel5 0.0,Channel6 0.0,Channel7 0.0,Channel8 0.0,BurnBackTime 0.0}
DECL FDAT FP44={TOOL_NO 1,BASE_NO 0,IPO_FRAME #BASE,POINT2[] " ",TQ_STATE FALSE}
DECL LDAT LCPDAT14={ACC 100.000,APO_DIST 100.000,APO_FAC 50.0000,AXIS_VEL 100.000,AXIS_ACC 100.000,ORI_TYP #VAR,CIRC_TYP #BASE,JERK_FAC 50.0000,GEAR_JERK 50.0000,EXAX_IGN 0}
DECL E6POS XP44={X 1502.02258,Y -578.292908,Z 1485.39441,A 30.5960255,B -59.1033821,C -140.023438,S 2,T 34,E1 180.000992,E2 179.999115,E3 180.003891,E4 0.0,E5 0.0,E6 0.0}
DECL E6POS XP45={X 1469.80408,Y -564.354736,Z 1523.67297,A 32.2780914,B -59.8028679,C -141.976486,S 2,T 34,E1 180.000992,E2 179.999115,E3 180.003891,E4 0.0,E5 0.0,E6 0.0}
DECL FDAT FP45={TOOL_NO 1,BASE_NO 0,IPO_FRAME #BASE,POINT2[] " ",TQ_STATE FALSE}
DECL PDAT PPDAT34={VEL 100.000,ACC 100.000,APO_DIST 100.000,GEAR_JERK 50.0000,EXAX_IGN 3}
DECL E6POS XP46={X 1469.80408,Y -564.354736,Z 1523.67297,A 32.2780914,B -59.8028679,C -141.976486,S 2,T 34,E1 180.000992,E2 179.999115,E3 180.003891,E4 0.0,E5 0.0,E6 0.0}
DECL FDAT FP46={TOOL_NO 1,BASE_NO 0,IPO_FRAME #BASE,POINT2[] " ",TQ_STATE FALSE}
DECL PDAT PPDAT35={VEL 100.000,ACC 100.000,APO_DIST 100.000,GEAR_JERK 50.0000,EXAX_IGN 3}
DECL ATBg_Start_T AS_WDAT25={JobModeId 1306102413,ParamSetId -1047099609,StartTime 0.0,PreFlowTime 0.0,Channel1 0.0,Channel2 2.00000,Channel3 0.0,Channel4 0.0,Channel5 0.0,Channel6 0.0,Channel7 0.0,Channel8 0.0,PurgeTime 0.0}
DECL ATBg_Weld_T AW_WDAT25={JobModeId -187662529,ParamSetId -430485013,Velocity 0.00830000,Channel1 30.0000,Channel2 1.00000,Channel3 0.0,Channel4 0.0,Channel5 0.0,Channel6 0.0,Channel7 0.0,Channel8 0.0}
DECL WTCg_WeaveDefinition_T WV_WDAT25={Pattern #None,Length 4.00000,Amplitude 2.00000,Angle 0.0}
DECL FDAT FP47={TOOL_NO 1,BASE_NO 0,IPO_FRAME #BASE,POINT2[] " ",TQ_STATE FALSE}
DECL PDAT PPDAT36={ACC 100.000,APO_DIST 100.000,APO_MODE #CPTP,GEAR_JERK 50.0000}
DECL E6POS XP47={X 1496.14221,Y -641.526245,Z 1369.59412,A -162.322510,B 68.5570297,C -52.6379738,S 2,T 2,E1 180.000992,E2 179.999115,E3 180.003891,E4 0.0,E5 0.0,E6 0.0}
DECL ATBg_Crater_T AC_WDAT26={JobModeId -187662529,ParamSetId -1375177600,CraterTime 0.100000,PostflowTime 0.100000,Channel1 30.0000,Channel2 1.00000,Channel3 0.0,Channel4 0.0,Channel5 0.0,Channel6 0.0,Channel7 0.0,Channel8 0.0,BurnBackTime 0.0}
DECL FDAT FP48={TOOL_NO 1,BASE_NO 0,IPO_FRAME #BASE,POINT2[] " ",TQ_STATE FALSE}
DECL LDAT LCPDAT15={ACC 100.000,APO_DIST 100.000,APO_FAC 50.0000,AXIS_VEL 100.000,AXIS_ACC 100.000,ORI_TYP #VAR,CIRC_TYP #BASE,JERK_FAC 50.0000,GEAR_JERK 50.0000,EXAX_IGN 0}
DECL E6POS XP48={X 1496.14221,Y -641.526245,Z 1369.59412,A -162.322510,B 68.5570297,C -52.6379738,S 2,T 2,E1 180.000992,E2 179.999115,E3 180.003891,E4 0.0,E5 0.0,E6 0.0}
DECL E6POS XP49={X 1448.11340,Y -622.753418,Z 1447.66052,A -156.764099,B 70.8568649,C -46.7135544,S 2,T 2,E1 180.000992,E2 179.999115,E3 180.003891,E4 0.0,E5 0.0,E6 0.0}
DECL FDAT FP49={TOOL_NO 1,BASE_NO 0,IPO_FRAME #BASE,POINT2[] " ",TQ_STATE FALSE}
DECL PDAT PPDAT37={VEL 100.000,ACC 100.000,APO_DIST 100.000,GEAR_JERK 50.0000,EXAX_IGN 3}
DECL E6POS XP50={X 1448.11340,Y -622.753418,Z 1447.66052,A -156.764099,B 70.8568649,C -46.7135544,S 2,T 2,E1 180.000992,E2 179.999115,E3 180.003891,E4 0.0,E5 0.0,E6 0.0}
DECL FDAT FP50={TOOL_NO 1,BASE_NO 0,IPO_FRAME #BASE,POINT2[] " ",TQ_STATE FALSE}
DECL PDAT PPDAT38={VEL 100.000,ACC 100.000,APO_DIST 100.000,GEAR_JERK 50.0000,EXAX_IGN 3}
DECL E6POS XP51={X 1485.35083,Y -636.504089,Z 1557.27551,A -66.0490341,B 70.7464371,C 47.0452,S 2,T 2,E1 180.000992,E2 179.999115,E3 180.003891,E4 0.0,E5 0.0,E6 0.0}
DECL FDAT FP51={TOOL_NO 1,BASE_NO 0,IPO_FRAME #BASE,POINT2[] " ",TQ_STATE FALSE}
DECL PDAT PPDAT39={VEL 100.000,ACC 100.000,APO_DIST 100.000,GEAR_JERK 50.0000,EXAX_IGN 3}
DECL ATBg_Start_T AS_WDAT27={JobModeId 1306102413,ParamSetId -1047099609,StartTime 0.0,PreFlowTime 0.0,Channel1 0.0,Channel2 2.00000,Channel3 0.0,Channel4 0.0,Channel5 0.0,Channel6 0.0,Channel7 0.0,Channel8 0.0,PurgeTime 0.0}
DECL ATBg_Weld_T AW_WDAT27={JobModeId -187662529,ParamSetId -430485013,Velocity 0.00830000,Channel1 30.0000,Channel2 1.00000,Channel3 0.0,Channel4 0.0,Channel5 0.0,Channel6 0.0,Channel7 0.0,Channel8 0.0}
DECL WTCg_WeaveDefinition_T WV_WDAT27={Pattern #None,Length 4.00000,Amplitude 2.00000,Angle 0.0}
DECL FDAT FP52={TOOL_NO 1,BASE_NO 0,IPO_FRAME #BASE,POINT2[] " ",TQ_STATE FALSE}
DECL PDAT PPDAT40={ACC 100.000,APO_DIST 100.000,APO_MODE #CPTP,GEAR_JERK 50.0000}
DECL E6POS XP52={X 1397.64026,Y -887.686279,Z 1403.38208,A -132.315063,B 46.3046303,C -23.7647057,S 2,T 10,E1 180.000992,E2 179.999115,E3 180.003891,E4 0.0,E5 0.0,E6 0.0}
DECL ATBg_Crater_T AC_WDAT28={JobModeId -187662529,ParamSetId -1375177600,CraterTime 0.100000,PostflowTime 0.100000,Channel1 30.0000,Channel2 1.00000,Channel3 0.0,Channel4 0.0,Channel5 0.0,Channel6 0.0,Channel7 0.0,Channel8 0.0,BurnBackTime 0.0}
DECL FDAT FP53={TOOL_NO 1,BASE_NO 0,IPO_FRAME #BASE,POINT2[] " ",TQ_STATE FALSE}
DECL LDAT LCPDAT16={ACC 100.000,APO_DIST 100.000,APO_FAC 50.0000,AXIS_VEL 100.000,AXIS_ACC 100.000,ORI_TYP #VAR,CIRC_TYP #BASE,JERK_FAC 50.0000,GEAR_JERK 50.0000,EXAX_IGN 0}
DECL E6POS XP53={X 1397.64026,Y -887.686279,Z 1403.38208,A -132.315063,B 46.3046303,C -23.7647057,S 2,T 10,E1 180.000992,E2 179.999115,E3 180.003891,E4 0.0,E5 0.0,E6 0.0}
DECL E6POS XP54={X 1367.67041,Y -870.237061,Z 1466.93665,A -128.024780,B 47.0159798,C -17.8683281,S 0,T 10,E1 180.000992,E2 179.999115,E3 180.003891,E4 0.0,E5 0.0,E6 0.0}
DECL FDAT FP54={TOOL_NO 1,BASE_NO 0,IPO_FRAME #BASE,POINT2[] " ",TQ_STATE FALSE}
DECL PDAT PPDAT41={VEL 100.000,ACC 100.000,APO_DIST 100.000,GEAR_JERK 50.0000,EXAX_IGN 3}
DECL ATBg_Start_T AS_WDAT29={JobModeId 1306102413,ParamSetId -1047099609,StartTime 0.0,PreFlowTime 0.0,Channel1 0.0,Channel2 2.00000,Channel3 0.0,Channel4 0.0,Channel5 0.0,Channel6 0.0,Channel7 0.0,Channel8 0.0,PurgeTime 0.0}
DECL ATBg_Weld_T AW_WDAT29={JobModeId -187662529,ParamSetId -430485013,Velocity 0.00830000,Channel1 30.0000,Channel2 1.00000,Channel3 0.0,Channel4 0.0,Channel5 0.0,Channel6 0.0,Channel7 0.0,Channel8 0.0}
DECL WTCg_WeaveDefinition_T WV_WDAT29={Pattern #None,Length 4.00000,Amplitude 2.00000,Angle 0.0}
DECL FDAT FP55={TOOL_NO 1,BASE_NO 0,IPO_FRAME #BASE,POINT2[] " ",TQ_STATE FALSE}
DECL PDAT PPDAT42={ACC 100.000,APO_DIST 100.000,APO_MODE #CPTP,GEAR_JERK 50.0000}
DECL E6POS XP55={X 1401.66064,Y -880.717651,Z 1461.76392,A 27.0726395,B -50.4124107,C -139.649567,S 2,T 42,E1 180.000992,E2 179.999115,E3 180.003891,E4 0.0,E5 0.0,E6 0.0}
DECL ATBg_Crater_T AC_WDAT30={JobModeId -187662529,ParamSetId -1375177600,CraterTime 0.100000,PostflowTime 0.100000,Channel1 30.0000,Channel2 1.00000,Channel3 0.0,Channel4 0.0,Channel5 0.0,Channel6 0.0,Channel7 0.0,Channel8 0.0,BurnBackTime 0.0}
DECL FDAT FP56={TOOL_NO 1,BASE_NO 0,IPO_FRAME #BASE,POINT2[] " ",TQ_STATE FALSE}
DECL LDAT LCPDAT17={ACC 100.000,APO_DIST 100.000,APO_FAC 50.0000,AXIS_VEL 100.000,AXIS_ACC 100.000,ORI_TYP #VAR,CIRC_TYP #BASE,JERK_FAC 50.0000,GEAR_JERK 50.0000,EXAX_IGN 0}
DECL E6POS XP56={X 1401.66064,Y -880.717651,Z 1461.76392,A 27.0726395,B -50.4124107,C -139.649567,S 2,T 42,E1 180.000992,E2 179.999115,E3 180.003891,E4 0.0,E5 0.0,E6 0.0}
DECL E6POS XP57={X 1369.23242,Y -857.527100,Z 1510.72119,A 28.6490726,B -51.0569115,C -141.685608,S 2,T 42,E1 180.000992,E2 179.999115,E3 180.003891,E4 0.0,E5 0.0,E6 0.0}
DECL FDAT FP57={TOOL_NO 1,BASE_NO 0,IPO_FRAME #BASE,POINT2[] " ",TQ_STATE FALSE}
DECL PDAT PPDAT43={VEL 100.000,ACC 100.000,APO_DIST 100.000,GEAR_JERK 50.0000,EXAX_IGN 3}
DECL E6POS XP58={X 1367.67041,Y -870.237061,Z 1466.93665,A -128.024780,B 47.0159798,C -17.8683281,S 0,T 10,E1 180.000992,E2 179.999115,E3 180.003891,E4 0.0,E5 0.0,E6 0.0}
DECL FDAT FP58={TOOL_NO 1,BASE_NO 0,IPO_FRAME #BASE,POINT2[] " ",TQ_STATE FALSE}
DECL PDAT PPDAT44={VEL 100.000,ACC 100.000,APO_DIST 100.000,GEAR_JERK 50.0000,EXAX_IGN 3}
DECL E6POS XP59={X 1369.23242,Y -857.527161,Z 1510.72119,A 28.6490707,B -51.0569115,C -141.685608,S 2,T 42,E1 180.000992,E2 179.999115,E3 180.003891,E4 0.0,E5 0.0,E6 0.0}
DECL FDAT FP59={TOOL_NO 1,BASE_NO 0,IPO_FRAME #BASE,POINT2[] " ",TQ_STATE FALSE}
DECL PDAT PPDAT45={VEL 100.000,ACC 100.000,APO_DIST 100.000,GEAR_JERK 50.0000,EXAX_IGN 3}
DECL E6POS XP60={X 945.867493,Y -554.763306,Z 2002.88318,A 61.1196899,B -55.2592354,C 178.350220,S 2,T 42,E1 67.5795670,E2 179.999115,E3 180.003891,E4 0.0,E5 0.0,E6 0.0}
DECL FDAT FP60={TOOL_NO 1,BASE_NO 0,IPO_FRAME #BASE,POINT2[] " ",TQ_STATE FALSE}
DECL PDAT PPDAT46={VEL 100.000,ACC 100.000,APO_DIST 100.000,GEAR_JERK 50.0000,EXAX_IGN 3}
DECL ATBg_Start_T AS_WDAT31={JobModeId 1306102413,ParamSetId -1047099609,StartTime 0.0,PreFlowTime 0.0,Channel1 0.0,Channel2 2.00000,Channel3 0.0,Channel4 0.0,Channel5 0.0,Channel6 0.0,Channel7 0.0,Channel8 0.0,PurgeTime 0.0}
DECL ATBg_Weld_T AW_WDAT31={JobModeId -187662529,ParamSetId -430485013,Velocity 0.00830000,Channel1 30.0000,Channel2 1.00000,Channel3 0.0,Channel4 0.0,Channel5 0.0,Channel6 0.0,Channel7 0.0,Channel8 0.0}
DECL WTCg_WeaveDefinition_T WV_WDAT31={Pattern #None,Length 4.00000,Amplitude 2.00000,Angle 0.0}
DECL FDAT FP61={TOOL_NO 1,BASE_NO 0,IPO_FRAME #BASE,POINT2[] " ",TQ_STATE FALSE}
DECL PDAT PPDAT47={ACC 100.000,APO_DIST 100.000,APO_MODE #CPTP,GEAR_JERK 50.0000}
DECL E6POS XP61={X 1418.66992,Y -837.542297,Z 1423.39563,A 44.6811409,B 77.4539,C 162.367722,S 2,T 42,E1 43.6475182,E2 179.999115,E3 180.003891,E4 0.0,E5 0.0,E6 0.0}
DECL ATBg_Crater_T AC_WDAT32={JobModeId -187662529,ParamSetId -1375177600,CraterTime 0.100000,PostflowTime 0.100000,Channel1 30.0000,Channel2 1.00000,Channel3 0.0,Channel4 0.0,Channel5 0.0,Channel6 0.0,Channel7 0.0,Channel8 0.0,BurnBackTime 0.0}
DECL FDAT FP62={TOOL_NO 1,BASE_NO 0,IPO_FRAME #BASE,POINT2[] " ",TQ_STATE FALSE}
DECL LDAT LCPDAT18={ACC 100.000,APO_DIST 100.000,APO_FAC 50.0000,AXIS_VEL 100.000,AXIS_ACC 100.000,ORI_TYP #VAR,CIRC_TYP #BASE,JERK_FAC 50.0000,GEAR_JERK 50.0000,EXAX_IGN 0}
DECL E6POS XP62={X 1418.66992,Y -837.542297,Z 1423.39563,A 44.6811409,B 77.4539,C 162.367722,S 2,T 42,E1 43.6475182,E2 179.999115,E3 180.003891,E4 0.0,E5 0.0,E6 0.0}
DECL E6POS XP63={X 1393.08484,Y -828.918091,Z 1461.18823,A 38.6596642,B 77.0320206,C 156.395554,S 2,T 42,E1 43.6475182,E2 179.999115,E3 180.003891,E4 0.0,E5 0.0,E6 0.0}
DECL FDAT FP63={TOOL_NO 1,BASE_NO 0,IPO_FRAME #BASE,POINT2[] " ",TQ_STATE FALSE}
DECL PDAT PPDAT48={VEL 100.000,ACC 100.000,APO_DIST 100.000,GEAR_JERK 50.0000,EXAX_IGN 3}
DECL E6POS XP64={X 1391.40466,Y -519.759521,Z 1528.67529,A 54.1671753,B 77.4182434,C 161.760574,S 2,T 42,E1 43.6475182,E2 179.999115,E3 180.003891,E4 0.0,E5 0.0,E6 0.0}
DECL FDAT FP64={TOOL_NO 1,BASE_NO 0,IPO_FRAME #BASE,POINT2[] " ",TQ_STATE FALSE}
DECL PDAT PPDAT49={VEL 100.000,ACC 100.000,APO_DIST 100.000,GEAR_JERK 50.0000,EXAX_IGN 3}
DECL E6POS XP65={X 1393.08484,Y -828.918091,Z 1461.18823,A 38.6596718,B 77.0320206,C 156.395554,S 2,T 42,E1 43.6475182,E2 179.999115,E3 180.003891,E4 0.0,E5 0.0,E6 0.0}
DECL FDAT FP65={TOOL_NO 1,BASE_NO 0,IPO_FRAME #BASE,POINT2[] " ",TQ_STATE FALSE}
DECL PDAT PPDAT50={VEL 100.000,ACC 100.000,APO_DIST 100.000,GEAR_JERK 50.0000,EXAX_IGN 3}
DECL E6POS XP66={X 1413.07727,Y -617.876160,Z 1470.88220,A 59.8442421,B 77.7953720,C 170.783493,S 2,T 42,E1 43.6475182,E2 179.999115,E3 180.003891,E4 0.0,E5 0.0,E6 0.0}
DECL FDAT FP66={TOOL_NO 1,BASE_NO 0,IPO_FRAME #BASE,POINT2[] " ",TQ_STATE FALSE}
DECL PDAT PPDAT51={VEL 100.000,ACC 100.000,APO_DIST 100.000,GEAR_JERK 50.0000,EXAX_IGN 3}
DECL ATBg_Start_T AS_WDAT33={JobModeId 1306102413,ParamSetId -1047099609,StartTime 0.0,PreFlowTime 0.0,Channel1 0.0,Channel2 2.00000,Channel3 0.0,Channel4 0.0,Channel5 0.0,Channel6 0.0,Channel7 0.0,Channel8 0.0,PurgeTime 0.0}
DECL ATBg_Weld_T AW_WDAT33={JobModeId -187662529,ParamSetId -430485013,Velocity 0.00830000,Channel1 30.0000,Channel2 1.00000,Channel3 0.0,Channel4 0.0,Channel5 0.0,Channel6 0.0,Channel7 0.0,Channel8 0.0}
DECL WTCg_WeaveDefinition_T WV_WDAT33={Pattern #None,Length 4.00000,Amplitude 2.00000,Angle 0.0}
DECL FDAT FP67={TOOL_NO 1,BASE_NO 0,IPO_FRAME #BASE,POINT2[] " ",TQ_STATE FALSE}
DECL PDAT PPDAT52={ACC 100.000,APO_DIST 100.000,APO_MODE #CPTP,GEAR_JERK 50.0000}
DECL E6POS XP67={X 1516.23657,Y -542.109131,Z 1407.86389,A 70.5701447,B 77.8772049,C 177.723236,S 2,T 42,E1 39.6729126,E2 179.999115,E3 180.003891,E4 0.0,E5 0.0,E6 0.0}
DECL ATBg_Crater_T AC_WDAT34={JobModeId -187662529,ParamSetId -1375177600,CraterTime 0.100000,PostflowTime 0.100000,Channel1 30.0000,Channel2 1.00000,Channel3 0.0,Channel4 0.0,Channel5 0.0,Channel6 0.0,Channel7 0.0,Channel8 0.0,BurnBackTime 0.0}
DECL FDAT FP68={TOOL_NO 1,BASE_NO 0,IPO_FRAME #BASE,POINT2[] " ",TQ_STATE FALSE}
DECL LDAT LCPDAT19={ACC 100.000,APO_DIST 100.000,APO_FAC 50.0000,AXIS_VEL 100.000,AXIS_ACC 100.000,ORI_TYP #VAR,CIRC_TYP #BASE,JERK_FAC 50.0000,GEAR_JERK 50.0000,EXAX_IGN 0}
DECL E6POS XP68={X 1516.23657,Y -542.109131,Z 1407.86389,A 70.5701447,B 77.8772049,C 177.723236,S 2,T 42,E1 39.6729126,E2 179.999115,E3 180.003891,E4 0.0,E5 0.0,E6 0.0}
DECL E6POS XP69={X 1382.02527,Y -494.258209,Z 1553.51624,A 50.0575943,B 77.0593185,C 156.721603,S 2,T 42,E1 39.6729126,E2 179.999115,E3 180.003891,E4 0.0,E5 0.0,E6 0.0}
DECL FDAT FP69={TOOL_NO 1,BASE_NO 0,IPO_FRAME #BASE,POINT2[] " ",TQ_STATE FALSE}
DECL PDAT PPDAT53={VEL 100.000,ACC 100.000,APO_DIST 100.000,GEAR_JERK 50.0000,EXAX_IGN 3}
DECL ATBg_Start_T AS_WDAT35={JobModeId 1306102413,ParamSetId -1047099609,StartTime 0.0,PreFlowTime 0.0,Channel1 0.0,Channel2 2.00000,Channel3 0.0,Channel4 0.0,Channel5 0.0,Channel6 0.0,Channel7 0.0,Channel8 0.0,PurgeTime 0.0}
DECL ATBg_Weld_T AW_WDAT35={JobModeId -187662529,ParamSetId -430485013,Velocity 0.00830000,Channel1 30.0000,Channel2 1.00000,Channel3 0.0,Channel4 0.0,Channel5 0.0,Channel6 0.0,Channel7 0.0,Channel8 0.0}
DECL WTCg_WeaveDefinition_T WV_WDAT35={Pattern #None,Length 4.00000,Amplitude 2.00000,Angle 0.0}
DECL FDAT FP70={TOOL_NO 1,BASE_NO 0,IPO_FRAME #BASE,POINT2[] " ",TQ_STATE FALSE}
DECL PDAT PPDAT54={ACC 100.000,APO_DIST 100.000,APO_MODE #CPTP,GEAR_JERK 50.0000}
DECL E6POS XP70={X 1579.26611,Y -136.946945,Z 1436.00012,A -88.2805939,B 58.3568497,C 3.02447629,S 2,T 10,E1 35.4823723,E2 180.095947,E3 180.003891,E4 0.0,E5 0.0,E6 0.0}
DECL ATBg_Crater_T AC_WDAT36={JobModeId -187662529,ParamSetId -1375177600,CraterTime 0.100000,PostflowTime 0.100000,Channel1 30.0000,Channel2 1.00000,Channel3 0.0,Channel4 0.0,Channel5 0.0,Channel6 0.0,Channel7 0.0,Channel8 0.0,BurnBackTime 0.0}
DECL FDAT FP71={TOOL_NO 1,BASE_NO 0,IPO_FRAME #BASE,POINT2[] " ",TQ_STATE FALSE}
DECL LDAT LCPDAT20={ACC 100.000,APO_DIST 100.000,APO_FAC 50.0000,AXIS_VEL 100.000,AXIS_ACC 100.000,ORI_TYP #VAR,CIRC_TYP #BASE,JERK_FAC 50.0000,GEAR_JERK 50.0000,EXAX_IGN 0}
DECL E6POS XP71={X 1579.26611,Y -136.946945,Z 1436.00012,A -88.2805939,B 58.3568497,C 3.02447629,S 2,T 10,E1 35.4823723,E2 180.095947,E3 180.003891,E4 0.0,E5 0.0,E6 0.0}
DECL E6POS XP72={X 1415.25378,Y -117.767067,Z 1567.15686,A -96.8179398,B 59.2228050,C -10.1517134,S 2,T 10,E1 35.4823723,E2 180.095947,E3 180.003891,E4 0.0,E5 0.0,E6 0.0}
DECL FDAT FP72={TOOL_NO 1,BASE_NO 0,IPO_FRAME #BASE,POINT2[] " ",TQ_STATE FALSE}
DECL PDAT PPDAT55={VEL 100.000,ACC 100.000,APO_DIST 100.000,GEAR_JERK 50.0000,EXAX_IGN 3}
DECL E6POS XP73={X 1415.25378,Y -117.767067,Z 1567.15686,A -96.8179398,B 59.2228050,C -10.1517162,S 2,T 10,E1 35.4823723,E2 180.095947,E3 180.003891,E4 0.0,E5 0.0,E6 0.0}
DECL FDAT FP73={TOOL_NO 1,BASE_NO 0,IPO_FRAME #BASE,POINT2[] " ",TQ_STATE FALSE}
DECL PDAT PPDAT56={VEL 100.000,ACC 100.000,APO_DIST 100.000,GEAR_JERK 50.0000,EXAX_IGN 3}
DECL ATBg_Start_T AS_WDAT37={JobModeId 1306102413,ParamSetId -1047099609,StartTime 0.0,PreFlowTime 0.0,Channel1 0.0,Channel2 2.00000,Channel3 0.0,Channel4 0.0,Channel5 0.0,Channel6 0.0,Channel7 0.0,Channel8 0.0,PurgeTime 0.0}
DECL ATBg_Weld_T AW_WDAT37={JobModeId -187662529,ParamSetId -430485013,Velocity 0.00830000,Channel1 30.0000,Channel2 1.00000,Channel3 0.0,Channel4 0.0,Channel5 0.0,Channel6 0.0,Channel7 0.0,Channel8 0.0}
DECL WTCg_WeaveDefinition_T WV_WDAT37={Pattern #None,Length 4.00000,Amplitude 2.00000,Angle 0.0}
DECL FDAT FP74={TOOL_NO 1,BASE_NO 0,IPO_FRAME #BASE,POINT2[] " ",TQ_STATE FALSE}
DECL PDAT PPDAT57={ACC 100.000,APO_DIST 100.000,APO_MODE #CPTP,GEAR_JERK 50.0000}
DECL E6POS XP74={X 1584.38623,Y 111.410187,Z 1386.96509,A 102.267334,B 52.8598785,C -171.791306,S 2,T 43,E1 30.6981010,E2 180.095947,E3 180.003891,E4 0.0,E5 0.0,E6 0.0}
DECL ATBg_Crater_T AC_WDAT38={JobModeId -187662529,ParamSetId -1375177600,CraterTime 0.100000,PostflowTime 0.100000,Channel1 30.0000,Channel2 1.00000,Channel3 0.0,Channel4 0.0,Channel5 0.0,Channel6 0.0,Channel7 0.0,Channel8 0.0,BurnBackTime 0.0}
DECL FDAT FP75={TOOL_NO 1,BASE_NO 0,IPO_FRAME #BASE,POINT2[] " ",TQ_STATE FALSE}
DECL LDAT LCPDAT21={ACC 100.000,APO_DIST 100.000,APO_FAC 50.0000,AXIS_VEL 100.000,AXIS_ACC 100.000,ORI_TYP #VAR,CIRC_TYP #BASE,JERK_FAC 50.0000,GEAR_JERK 50.0000,EXAX_IGN 0}
DECL E6POS XP75={X 1584.38623,Y 111.410187,Z 1386.96509,A 102.267334,B 52.8598785,C -171.791306,S 2,T 43,E1 30.6981010,E2 180.095947,E3 180.003891,E4 0.0,E5 0.0,E6 0.0}
DECL E6POS XP76={X 1441.27734,Y -90.4894485,Z 1536.43652,A -100.739212,B 68.4979858,C -14.1514530,S 2,T 10,E1 34.8087654,E2 180.095947,E3 180.003891,E4 0.0,E5 0.0,E6 0.0}
DECL FDAT FP76={TOOL_NO 1,BASE_NO 0,IPO_FRAME #BASE,POINT2[] " ",TQ_STATE FALSE}
DECL PDAT PPDAT58={VEL 100.000,ACC 100.000,APO_DIST 100.000,GEAR_JERK 50.0000,EXAX_IGN 3}
DECL E6POS XP77={X 1472.05359,Y -555.361511,Z 1447.94543,A 53.5533104,B 56.5259285,C 162.220825,S 2,T 42,E1 180.000992,E2 179.999115,E3 180.003891,E4 0.0,E5 0.0,E6 0.0}
DECL FDAT FP77={TOOL_NO 1,BASE_NO 0,IPO_FRAME #BASE,POINT2[] " ",TQ_STATE FALSE}
DECL PDAT PPDAT59={VEL 100.000,ACC 100.000,APO_DIST 100.000,GEAR_JERK 50.0000,EXAX_IGN 3}
DECL ATBg_Start_T AS_WDAT39={JobModeId 1306102413,ParamSetId -1047099609,StartTime 0.0,PreFlowTime 0.0,Channel1 0.0,Channel2 2.00000,Channel3 0.0,Channel4 0.0,Channel5 0.0,Channel6 0.0,Channel7 0.0,Channel8 0.0,PurgeTime 0.0}
DECL ATBg_Weld_T AW_WDAT39={JobModeId 1306102413,ParamSetId -540622874,Velocity 0.00830000,Channel1 0.0,Channel2 1.00000,Channel3 0.0,Channel4 0.0,Channel5 0.0,Channel6 0.0,Channel7 0.0,Channel8 0.0}
DECL WTCg_WeaveDefinition_T WV_WDAT39={Pattern #None,Length 4.00000,Amplitude 2.00000,Angle 0.0}
DECL FDAT FP78={TOOL_NO 1,BASE_NO 0,IPO_FRAME #BASE,POINT2[] " ",TQ_STATE FALSE}
DECL PDAT PPDAT60={ACC 100.000,APO_DIST 100.000,APO_MODE #CPTP,GEAR_JERK 50.0000}
DECL E6POS XP78={X 1344.34131,Y 545.107666,Z 1613.57458,A 101.826927,B 70.2007828,C 176.589447,S 2,T 35,E1 229.997406,E2 195.002228,E3 195.004227,E4 0.0,E5 0.0,E6 0.0}
DECL ATBg_Crater_T AC_WDAT40={JobModeId -187662529,ParamSetId -1375177600,CraterTime 0.100000,PostflowTime 0.100000,Channel1 30.0000,Channel2 1.00000,Channel3 0.0,Channel4 0.0,Channel5 0.0,Channel6 0.0,Channel7 0.0,Channel8 0.0,BurnBackTime 0.0}
DECL FDAT FP79={TOOL_NO 1,BASE_NO 0,IPO_FRAME #BASE,POINT2[] " ",TQ_STATE FALSE}
DECL LDAT LCPDAT22={ACC 100.000,APO_DIST 100.000,APO_FAC 50.0000,AXIS_VEL 100.000,AXIS_ACC 100.000,ORI_TYP #VAR,CIRC_TYP #BASE,JERK_FAC 50.0000,GEAR_JERK 50.0000,EXAX_IGN 0}
DECL E6POS XP79={X 1345.37646,Y 533.994629,Z 1613.35364,A 102.084946,B 70.2269897,C 176.990280,S 2,T 35,E1 229.997406,E2 195.002228,E3 195.004227,E4 0.0,E5 0.0,E6 0.0}
DECL ATBg_Start_T AS_WDAT41={JobModeId -187662529,ParamSetId 687014726,StartTime 0.0,PreFlowTime 0.100000,Channel1 30.0000,Channel2 1.00000,Channel3 0.0,Channel4 0.0,Channel5 0.0,Channel6 0.0,Channel7 0.0,Channel8 0.0,PurgeTime 0.0}
DECL ATBg_Weld_T AW_WDAT41={JobModeId -187662529,ParamSetId -430485013,Velocity 0.00830000,Channel1 30.0000,Channel2 1.00000,Channel3 0.0,Channel4 0.0,Channel5 0.0,Channel6 0.0,Channel7 0.0,Channel8 0.0}
DECL WTCg_WeaveDefinition_T WV_WDAT41={Pattern #None,Length 4.00000,Amplitude 2.00000,Angle 0.0}
DECL FDAT FP80={TOOL_NO 1,BASE_NO 0,IPO_FRAME #BASE,POINT2[] " ",TQ_STATE FALSE}
DECL PDAT PPDAT61={ACC 100.000,APO_DIST 100.000,APO_MODE #CPTP,GEAR_JERK 50.0000}
DECL E6POS XP80={X 1389.51404,Y 302.941376,Z 1610.34790,A 104.640984,B 74.7491074,C -177.070221,S 2,T 35,E1 229.997360,E2 195.002197,E3 195.004211,E4 0.0,E5 0.0,E6 0.0}
DECL ATBg_Crater_T AC_WDAT42={JobModeId -187662529,ParamSetId -1375177600,CraterTime 0.100000,PostflowTime 0.100000,Channel1 30.0000,Channel2 1.00000,Channel3 0.0,Channel4 0.0,Channel5 0.0,Channel6 0.0,Channel7 0.0,Channel8 0.0,BurnBackTime 0.0}
DECL FDAT FP81={TOOL_NO 1,BASE_NO 0,IPO_FRAME #BASE,POINT2[] " ",TQ_STATE FALSE}
DECL LDAT LCPDAT23={ACC 100.000,APO_DIST 100.000,APO_FAC 50.0000,AXIS_VEL 100.000,AXIS_ACC 100.000,ORI_TYP #VAR,CIRC_TYP #BASE,JERK_FAC 50.0000,GEAR_JERK 50.0000,EXAX_IGN 0}
DECL E6POS XP81={X 1391.36011,Y 294.178101,Z 1611.30188,A 106.205254,B 80.0392685,C -175.542023,S 2,T 35,E1 229.997360,E2 195.002197,E3 195.004211,E4 0.0,E5 0.0,E6 0.0}
DECL ATBg_Start_T AS_WDAT43={JobModeId -187662529,ParamSetId 687014726,StartTime 0.0,PreFlowTime 0.100000,Channel1 30.0000,Channel2 1.00000,Channel3 0.0,Channel4 0.0,Channel5 0.0,Channel6 0.0,Channel7 0.0,Channel8 0.0,PurgeTime 0.0}
DECL ATBg_Weld_T AW_WDAT43={JobModeId -187662529,ParamSetId -430485013,Velocity 0.00830000,Channel1 30.0000,Channel2 1.00000,Channel3 0.0,Channel4 0.0,Channel5 0.0,Channel6 0.0,Channel7 0.0,Channel8 0.0}
DECL WTCg_WeaveDefinition_T WV_WDAT43={Pattern #None,Length 4.00000,Amplitude 2.00000,Angle 0.0}
DECL FDAT FP82={TOOL_NO 1,BASE_NO 0,IPO_FRAME #BASE,POINT2[] " ",TQ_STATE FALSE}
DECL PDAT PPDAT62={ACC 100.000,APO_DIST 100.000,APO_MODE #CPTP,GEAR_JERK 50.0000}
DECL E6POS XP82={X 1405.05640,Y -51.4842529,Z 1609.80847,A 140.270340,B 86.4778442,C -127.943268,S 2,T 34,E1 229.997360,E2 195.002197,E3 195.004211,E4 0.0,E5 0.0,E6 0.0}
DECL ATBg_Crater_T AC_WDAT44={JobModeId -187662529,ParamSetId -1375177600,CraterTime 0.100000,PostflowTime 0.100000,Channel1 30.0000,Channel2 1.00000,Channel3 0.0,Channel4 0.0,Channel5 0.0,Channel6 0.0,Channel7 0.0,Channel8 0.0,BurnBackTime 0.0}
DECL FDAT FP83={TOOL_NO 1,BASE_NO 0,IPO_FRAME #BASE,POINT2[] " ",TQ_STATE FALSE}
DECL LDAT LCPDAT24={ACC 100.000,APO_DIST 100.000,APO_FAC 50.0000,AXIS_VEL 100.000,AXIS_ACC 100.000,ORI_TYP #VAR,CIRC_TYP #BASE,JERK_FAC 50.0000,GEAR_JERK 50.0000,EXAX_IGN 0}
DECL E6POS XP83={X 1405.05640,Y -51.4842529,Z 1609.80847,A 140.270340,B 86.4778442,C -127.943268,S 2,T 34,E1 229.997360,E2 195.002197,E3 195.004211,E4 0.0,E5 0.0,E6 0.0}
DECL E6POS XP84={X 1399.90735,Y -51.4098587,Z 1616.55884,A 136.356430,B 86.7458420,C -131.864014,S 2,T 34,E1 229.997360,E2 195.002197,E3 195.004211,E4 0.0,E5 0.0,E6 0.0}
DECL FDAT FP84={TOOL_NO 1,BASE_NO 0,IPO_FRAME #BASE,POINT2[] " ",TQ_STATE FALSE}
DECL PDAT PPDAT63={VEL 100.000,ACC 100.000,APO_DIST 100.000,APO_MODE #CDIS,GEAR_JERK 50.0000,EXAX_IGN 3}
DECL E6POS XP85={X 1319.20300,Y -50.2438545,Z 1728.13440,A 26.8801632,B 85.2404327,C 118.532234,S 2,T 34,E1 229.997360,E2 195.002197,E3 195.004211,E4 0.0,E5 0.0,E6 0.0}
DECL FDAT FP85={TOOL_NO 1,BASE_NO 0,IPO_FRAME #BASE,POINT2[] " ",TQ_STATE FALSE}
DECL PDAT PPDAT64={VEL 100.000,ACC 100.000,APO_DIST 100.000,APO_MODE #CDIS,GEAR_JERK 50.0000,EXAX_IGN 3}
DECL E6POS XP86={X 1308.38721,Y -175.908188,Z 1728.13440,A 21.4040012,B 85.2404327,C 118.532234,S 2,T 34,E1 229.997360,E2 195.002197,E3 195.004211,E4 0.0,E5 0.0,E6 0.0}
DECL FDAT FP86={TOOL_NO 1,BASE_NO 0,IPO_FRAME #BASE,POINT2[] " ",TQ_STATE FALSE}
DECL PDAT PPDAT65={VEL 100.000,ACC 100.000,APO_DIST 100.000,APO_MODE #CDIS,GEAR_JERK 50.0000,EXAX_IGN 3}
DECL ATBg_Start_T AS_WDAT45={JobModeId -187662529,ParamSetId 687014726,StartTime 0.0,PreFlowTime 0.100000,Channel1 30.0000,Channel2 1.00000,Channel3 0.0,Channel4 0.0,Channel5 0.0,Channel6 0.0,Channel7 0.0,Channel8 0.0,PurgeTime 0.0}
DECL ATBg_Weld_T AW_WDAT45={JobModeId -187662529,ParamSetId -430485013,Velocity 0.00830000,Channel1 30.0000,Channel2 1.00000,Channel3 0.0,Channel4 0.0,Channel5 0.0,Channel6 0.0,Channel7 0.0,Channel8 0.0}
DECL WTCg_WeaveDefinition_T WV_WDAT45={Pattern #None,Length 4.00000,Amplitude 2.00000,Angle 0.0}
DECL FDAT FP87={TOOL_NO 1,BASE_NO 0,IPO_FRAME #BASE,POINT2[] " ",TQ_STATE FALSE}
DECL PDAT PPDAT66={ACC 100.000,APO_DIST 100.000,APO_MODE #CPTP,GEAR_JERK 50.0000}
DECL E6POS XP87={X 1397.26331,Y -207.500198,Z 1611.62207,A -136.868607,B 85.8667068,C -39.2035751,S 2,T 2,E1 229.997360,E2 195.002197,E3 195.004211,E4 0.0,E5 0.0,E6 0.0}
DECL ATBg_Crater_T AC_WDAT46={JobModeId -187662529,ParamSetId -1375177600,CraterTime 0.100000,PostflowTime 0.100000,Channel1 30.0000,Channel2 1.00000,Channel3 0.0,Channel4 0.0,Channel5 0.0,Channel6 0.0,Channel7 0.0,Channel8 0.0,BurnBackTime 0.0}
DECL FDAT FP88={TOOL_NO 1,BASE_NO 0,IPO_FRAME #BASE,POINT2[] " ",TQ_STATE FALSE}
DECL LDAT LCPDAT25={ACC 100.000,APO_DIST 100.000,APO_FAC 50.0000,AXIS_VEL 100.000,AXIS_ACC 100.000,ORI_TYP #VAR,CIRC_TYP #BASE,JERK_FAC 50.0000,GEAR_JERK 50.0000,EXAX_IGN 0}
DECL E6POS XP88={X 1397.26331,Y -207.500198,Z 1611.62207,A -136.868607,B 85.8667068,C -39.2035751,S 2,T 2,E1 229.997360,E2 195.002197,E3 195.004211,E4 0.0,E5 0.0,E6 0.0}
DECL E6POS XP89={X 1306.19275,Y -196.588913,Z 1703.97925,A -68.7830734,B 86.4150162,C 29.0020599,S 2,T 2,E1 229.997360,E2 195.002197,E3 195.004211,E4 0.0,E5 0.0,E6 0.0}
DECL FDAT FP89={TOOL_NO 1,BASE_NO 0,IPO_FRAME #BASE,POINT2[] " ",TQ_STATE FALSE}
DECL PDAT PPDAT67={VEL 100.000,ACC 100.000,APO_DIST 100.000,APO_MODE #CDIS,GEAR_JERK 50.0000,EXAX_IGN 3}
DECL ATBg_Start_T AS_WDAT47={JobModeId -187662529,ParamSetId 687014726,StartTime 0.0,PreFlowTime 0.100000,Channel1 30.0000,Channel2 1.00000,Channel3 0.0,Channel4 0.0,Channel5 0.0,Channel6 0.0,Channel7 0.0,Channel8 0.0,PurgeTime 0.0}
DECL ATBg_Weld_T AW_WDAT47={JobModeId -187662529,ParamSetId -430485013,Velocity 0.00830000,Channel1 30.0000,Channel2 1.00000,Channel3 0.0,Channel4 0.0,Channel5 0.0,Channel6 0.0,Channel7 0.0,Channel8 0.0}
DECL WTCg_WeaveDefinition_T WV_WDAT47={Pattern #None,Length 4.00000,Amplitude 2.00000,Angle 0.0}
DECL FDAT FP90={TOOL_NO 1,BASE_NO 0,IPO_FRAME #BASE,POINT2[] " ",TQ_STATE FALSE}
DECL PDAT PPDAT68={ACC 100.000,APO_DIST 100.000,APO_MODE #CPTP,GEAR_JERK 50.0000}
DECL E6POS XP90={X 1232.65955,Y -891.276917,Z 1635.28589,A -96.7124100,B 54.7162971,C 6.76454,S 2,T 10,E1 229.997360,E2 195.002197,E3 195.004211,E4 0.0,E5 0.0,E6 0.0}
DECL ATBg_Crater_T AC_WDAT48={JobModeId -187662529,ParamSetId -1375177600,CraterTime 0.100000,PostflowTime 0.100000,Channel1 30.0000,Channel2 1.00000,Channel3 0.0,Channel4 0.0,Channel5 0.0,Channel6 0.0,Channel7 0.0,Channel8 0.0,BurnBackTime 0.0}
DECL FDAT FP91={TOOL_NO 1,BASE_NO 0,IPO_FRAME #BASE,POINT2[] " ",TQ_STATE FALSE}
DECL LDAT LCPDAT26={ACC 100.000,APO_DIST 100.000,APO_FAC 50.0000,AXIS_VEL 100.000,AXIS_ACC 100.000,ORI_TYP #VAR,CIRC_TYP #BASE,JERK_FAC 50.0000,GEAR_JERK 50.0000,EXAX_IGN 0}
DECL E6POS XP91={X 1232.65955,Y -891.276917,Z 1635.28589,A -96.7124100,B 54.7162971,C 6.76454,S 2,T 10,E1 229.997360,E2 195.002197,E3 195.004211,E4 0.0,E5 0.0,E6 0.0}
DECL E6POS XP92={X 1054.34692,Y -757.859863,Z 1864.28418,A -84.9267426,B 47.8384056,C 21.8099632,S 2,T 10,E1 229.997360,E2 195.002197,E3 195.004211,E4 0.0,E5 0.0,E6 0.0}
DECL FDAT FP92={TOOL_NO 1,BASE_NO 0,IPO_FRAME #BASE,POINT2[] " ",TQ_STATE FALSE}
DECL PDAT PPDAT69={VEL 100.000,ACC 100.000,APO_DIST 100.000,APO_MODE #CDIS,GEAR_JERK 50.0000,EXAX_IGN 3}
DECL E6POS XP93={X 1192.32471,Y 472.459,Z 1776.73877,A 83.1334229,B 67.4761200,C 156.576218,S 2,T 35,E1 229.997406,E2 195.002228,E3 195.004227,E4 0.0,E5 0.0,E6 0.0}
DECL FDAT FP93={TOOL_NO 1,BASE_NO 0,IPO_FRAME #BASE,POINT2[] " ",TQ_STATE FALSE}
DECL PDAT PPDAT70={VEL 100.000,ACC 100.000,APO_DIST 100.000,APO_MODE #CDIS,GEAR_JERK 50.0000,EXAX_IGN 3}
DECL E6POS XP94={X 1203.56567,Y 245.655396,Z 1802.88013,A 72.3533630,B 68.4953918,C 154.352661,S 2,T 35,E1 229.997391,E2 195.002228,E3 195.004227,E4 0.0,E5 0.0,E6 0.0}
DECL FDAT FP94={TOOL_NO 1,BASE_NO 0,IPO_FRAME #BASE,POINT2[] " ",TQ_STATE FALSE}
DECL PDAT PPDAT71={VEL 100.000,ACC 100.000,APO_DIST 100.000,APO_MODE #CDIS,GEAR_JERK 50.0000,EXAX_IGN 3}
DECL E6POS XP95={X 1366.39880,Y 202.321213,Z 1652.72510,A 92.5657654,B 80.7616730,C 174.120758,S 2,T 35,E1 229.997360,E2 195.002197,E3 195.004211,E4 0.0,E5 0.0,E6 0.0}
DECL FDAT FP95={TOOL_NO 1,BASE_NO 0,IPO_FRAME #BASE,POINT2[] " ",TQ_STATE FALSE}
DECL PDAT PPDAT72={VEL 100.000,ACC 100.000,APO_DIST 100.000,APO_MODE #CDIS,GEAR_JERK 50.0000,EXAX_IGN 3}
DECL E6POS XP96={X 1171.60815,Y -889.236572,Z 1696.34497,A -96.0087738,B 50.3284950,C 9.56970692,S 2,T 10,E1 190.873,E2 195.002197,E3 195.004211,E4 0.0,E5 0.0,E6 0.0}
DECL FDAT FP96={TOOL_NO 1,BASE_NO 0,IPO_FRAME #BASE,POINT2[] " ",TQ_STATE FALSE}
DECL PDAT PPDAT73={VEL 100.000,ACC 100.000,APO_DIST 100.000,APO_MODE #CDIS,GEAR_JERK 50.0000,EXAX_IGN 3}
DECL ATBg_Start_T AS_WDAT49={JobModeId -187662529,ParamSetId 687014726,StartTime 0.0,PreFlowTime 0.100000,Channel1 30.0000,Channel2 1.00000,Channel3 0.0,Channel4 0.0,Channel5 0.0,Channel6 0.0,Channel7 0.0,Channel8 0.0,PurgeTime 0.0}
DECL ATBg_Weld_T AW_WDAT49={JobModeId -187662529,ParamSetId -430485013,Velocity 0.00830000,Channel1 30.0000,Channel2 1.00000,Channel3 0.0,Channel4 0.0,Channel5 0.0,Channel6 0.0,Channel7 0.0,Channel8 0.0}
DECL WTCg_WeaveDefinition_T WV_WDAT49={Pattern #None,Length 4.00000,Amplitude 2.00000,Angle 0.0}
DECL FDAT FP97={TOOL_NO 1,BASE_NO 0,IPO_FRAME #BASE,POINT2[] " ",TQ_STATE FALSE}
DECL PDAT PPDAT74={ACC 100.000,APO_DIST 100.000,APO_MODE #CPTP,GEAR_JERK 50.0000}
DECL E6POS XP97={X 1206.43689,Y -921.566711,Z 1635.16187,A -94.9919662,B 61.2246590,C 10.2442360,S 2,T 10,E1 190.873,E2 195.002197,E3 195.004211,E4 0.0,E5 0.0,E6 0.0}
DECL ATBg_Crater_T AC_WDAT50={JobModeId -187662529,ParamSetId -1375177600,CraterTime 0.100000,PostflowTime 0.100000,Channel1 30.0000,Channel2 1.00000,Channel3 0.0,Channel4 0.0,Channel5 0.0,Channel6 0.0,Channel7 0.0,Channel8 0.0,BurnBackTime 0.0}
DECL FDAT FP98={TOOL_NO 1,BASE_NO 0,IPO_FRAME #BASE,POINT2[] " ",TQ_STATE FALSE}
DECL LDAT LCPDAT27={ACC 100.000,APO_DIST 100.000,APO_FAC 50.0000,AXIS_VEL 100.000,AXIS_ACC 100.000,ORI_TYP #VAR,CIRC_TYP #BASE,JERK_FAC 50.0000,GEAR_JERK 50.0000,EXAX_IGN 0}
DECL E6POS XP98={X 1206.43689,Y -921.566711,Z 1635.16187,A -94.9919662,B 61.2246590,C 10.2442360,S 2,T 10,E1 190.873,E2 195.002197,E3 195.004211,E4 0.0,E5 0.0,E6 0.0}
DECL ATBg_Crater_T AC_WDAT51={JobModeId -187662529,ParamSetId -1375177600,CraterTime 0.100000,PostflowTime 0.100000,Channel1 30.0000,Channel2 1.00000,Channel3 0.0,Channel4 0.0,Channel5 0.0,Channel6 0.0,Channel7 0.0,Channel8 0.0,BurnBackTime 0.0}
DECL FDAT FP99={TOOL_NO 1,BASE_NO 0,IPO_FRAME #BASE,POINT2[] " ",TQ_STATE FALSE}
DECL LDAT LCPDAT28={ACC 100.000,APO_DIST 100.000,APO_FAC 50.0000,AXIS_VEL 100.000,AXIS_ACC 100.000,ORI_TYP #VAR,CIRC_TYP #BASE,JERK_FAC 50.0000,GEAR_JERK 50.0000,EXAX_IGN 0}
DECL E6POS XP99={X 1194.17407,Y -927.370056,Z 1636.72192,A -96.0782471,B 61.4487839,C 9.53255939,S 2,T 10,E1 190.873,E2 195.002197,E3 195.004211,E4 0.0,E5 0.0,E6 0.0}
DECL ATBg_Start_T AS_WDAT52={JobModeId -187662529,ParamSetId 687014726,StartTime 0.0,PreFlowTime 0.100000,Channel1 30.0000,Channel2 1.00000,Channel3 0.0,Channel4 0.0,Channel5 0.0,Channel6 0.0,Channel7 0.0,Channel8 0.0,PurgeTime 0.0}
DECL ATBg_Weld_T AW_WDAT52={JobModeId -187662529,ParamSetId -430485013,Velocity 0.00830000,Channel1 30.0000,Channel2 1.00000,Channel3 0.0,Channel4 0.0,Channel5 0.0,Channel6 0.0,Channel7 0.0,Channel8 0.0}
DECL WTCg_WeaveDefinition_T WV_WDAT52={Pattern #None,Length 4.00000,Amplitude 2.00000,Angle 0.0}
DECL FDAT FP100={TOOL_NO 1,BASE_NO 0,IPO_FRAME #BASE,POINT2[] " ",TQ_STATE FALSE}
DECL PDAT PPDAT75={ACC 100.000,APO_DIST 100.000,APO_MODE #CPTP,GEAR_JERK 50.0000}
DECL E6POS XP100={X 1254.47900,Y -806.532104,Z 1613.77075,A -96.0353394,B 70.1869659,C 2.27105737,S 2,T 10,E1 190.873,E2 195.002197,E3 195.004211,E4 0.0,E5 0.0,E6 0.0}
DECL ATBg_Crater_T AC_WDAT53={JobModeId -187662529,ParamSetId -1375177600,CraterTime 0.100000,PostflowTime 0.100000,Channel1 30.0000,Channel2 1.00000,Channel3 0.0,Channel4 0.0,Channel5 0.0,Channel6 0.0,Channel7 0.0,Channel8 0.0,BurnBackTime 0.0}
DECL FDAT FP101={TOOL_NO 1,BASE_NO 0,IPO_FRAME #BASE,POINT2[] " ",TQ_STATE FALSE}
DECL LDAT LCPDAT29={ACC 100.000,APO_DIST 100.000,APO_FAC 50.0000,AXIS_VEL 100.000,AXIS_ACC 100.000,ORI_TYP #VAR,CIRC_TYP #BASE,JERK_FAC 50.0000,GEAR_JERK 50.0000,EXAX_IGN 0}
DECL E6POS XP101={X 1253.55212,Y -812.493896,Z 1618.97900,A -96.4830627,B 65.4992599,C 1.85604811,S 2,T 10,E1 190.873,E2 195.002197,E3 195.004211,E4 0.0,E5 0.0,E6 0.0}
DECL ATBg_Start_T AS_WDAT54={JobModeId -187662529,ParamSetId 687014726,StartTime 0.0,PreFlowTime 0.100000,Channel1 30.0000,Channel2 1.00000,Channel3 0.0,Channel4 0.0,Channel5 0.0,Channel6 0.0,Channel7 0.0,Channel8 0.0,PurgeTime 0.0}
DECL ATBg_Weld_T AW_WDAT54={JobModeId -187662529,ParamSetId -430485013,Velocity 0.00830000,Channel1 30.0000,Channel2 1.00000,Channel3 0.0,Channel4 0.0,Channel5 0.0,Channel6 0.0,Channel7 0.0,Channel8 0.0}
DECL WTCg_WeaveDefinition_T WV_WDAT54={Pattern #None,Length 4.00000,Amplitude 2.00000,Angle 0.0}
DECL FDAT FP102={TOOL_NO 1,BASE_NO 0,IPO_FRAME #BASE,POINT2[] " ",TQ_STATE FALSE}
DECL PDAT PPDAT76={ACC 100.000,APO_DIST 100.000,APO_MODE #CPTP,GEAR_JERK 50.0000}
DECL E6POS XP102={X 1246.51099,Y -824.909851,Z 1637.50818,A -96.9019775,B 54.7476616,C 1.71330380,S 2,T 10,E1 190.873,E2 195.002197,E3 195.004211,E4 0.0,E5 0.0,E6 0.0}
DECL ATBg_Crater_T AC_WDAT55={JobModeId -187662529,ParamSetId -1375177600,CraterTime 0.100000,PostflowTime 0.100000,Channel1 30.0000,Channel2 1.00000,Channel3 0.0,Channel4 0.0,Channel5 0.0,Channel6 0.0,Channel7 0.0,Channel8 0.0,BurnBackTime 0.0}
DECL FDAT FP103={TOOL_NO 1,BASE_NO 0,IPO_FRAME #BASE,POINT2[] " ",TQ_STATE FALSE}
DECL LDAT LCPDAT30={ACC 100.000,APO_DIST 100.000,APO_FAC 50.0000,AXIS_VEL 100.000,AXIS_ACC 100.000,ORI_TYP #VAR,CIRC_TYP #BASE,JERK_FAC 50.0000,GEAR_JERK 50.0000,EXAX_IGN 0}
DECL E6POS XP103={X 1245.91785,Y -828.361267,Z 1642.64575,A -97.0760269,B 51.0904427,C 1.57438397,S 2,T 10,E1 190.873,E2 195.002197,E3 195.004211,E4 0.0,E5 0.0,E6 0.0}
DECL E6POS XP104={X 993.488,Y -653.571472,Z 1941.27576,A -82.8141479,B 41.6257553,C 21.1250896,S 2,T 10,E1 190.873,E2 195.002197,E3 195.004211,E4 0.0,E5 0.0,E6 0.0}
DECL FDAT FP104={TOOL_NO 1,BASE_NO 0,IPO_FRAME #BASE,POINT2[] " ",TQ_STATE FALSE}
DECL PDAT PPDAT77={VEL 100.000,ACC 100.000,APO_DIST 100.000,APO_MODE #CDIS,GEAR_JERK 50.0000,EXAX_IGN 3}
DECL ATBg_Start_T AS_WDAT56={JobModeId -187662529,ParamSetId 687014726,StartTime 0.0,PreFlowTime 0.100000,Channel1 30.0000,Channel2 1.00000,Channel3 0.0,Channel4 0.0,Channel5 0.0,Channel6 0.0,Channel7 0.0,Channel8 0.0,PurgeTime 0.0}
DECL ATBg_Weld_T AW_WDAT56={JobModeId -187662529,ParamSetId -430485013,Velocity 0.00830000,Channel1 30.0000,Channel2 1.00000,Channel3 0.0,Channel4 0.0,Channel5 0.0,Channel6 0.0,Channel7 0.0,Channel8 0.0}
DECL WTCg_WeaveDefinition_T WV_WDAT56={Pattern #None,Length 4.00000,Amplitude 2.00000,Angle 0.0}
DECL FDAT FP105={TOOL_NO 1,BASE_NO 0,IPO_FRAME #BASE,POINT2[] " ",TQ_STATE FALSE}
DECL PDAT PPDAT78={ACC 100.000,APO_DIST 100.000,APO_MODE #CPTP,GEAR_JERK 50.0000}
DECL E6POS XP105={X 1288.91138,Y -655.583923,Z 1673.83777,A -92.6688843,B 61.3095779,C 22.6213436,S 2,T 10,E1 190.873,E2 195.002197,E3 195.004211,E4 0.0,E5 0.0,E6 0.0}
DECL ATBg_Crater_T AC_WDAT57={JobModeId -187662529,ParamSetId -1375177600,CraterTime 0.100000,PostflowTime 0.100000,Channel1 30.0000,Channel2 1.00000,Channel3 0.0,Channel4 0.0,Channel5 0.0,Channel6 0.0,Channel7 0.0,Channel8 0.0,BurnBackTime 0.0}
DECL FDAT FP106={TOOL_NO 1,BASE_NO 0,IPO_FRAME #BASE,POINT2[] " ",TQ_STATE FALSE}
DECL LDAT LCPDAT31={ACC 100.000,APO_DIST 100.000,APO_FAC 50.0000,AXIS_VEL 100.000,AXIS_ACC 100.000,ORI_TYP #VAR,CIRC_TYP #BASE,JERK_FAC 50.0000,GEAR_JERK 50.0000,EXAX_IGN 0}
DECL E6POS XP106={X 1291.79114,Y -651.086548,Z 1668.95923,A -88.7677460,B 65.1891708,C 26.1072254,S 2,T 10,E1 190.873,E2 195.002197,E3 195.004211,E4 0.0,E5 0.0,E6 0.0}
DECL ATBg_Start_T AS_WDAT58={JobModeId -187662529,ParamSetId 687014726,StartTime 0.0,PreFlowTime 0.100000,Channel1 30.0000,Channel2 1.00000,Channel3 0.0,Channel4 0.0,Channel5 0.0,Channel6 0.0,Channel7 0.0,Channel8 0.0,PurgeTime 0.0}
DECL ATBg_Weld_T AW_WDAT58={JobModeId -187662529,ParamSetId -430485013,Velocity 0.00830000,Channel1 30.0000,Channel2 1.00000,Channel3 0.0,Channel4 0.0,Channel5 0.0,Channel6 0.0,Channel7 0.0,Channel8 0.0}
DECL WTCg_WeaveDefinition_T WV_WDAT58={Pattern #None,Length 4.00000,Amplitude 2.00000,Angle 0.0}
DECL FDAT FP107={TOOL_NO 1,BASE_NO 0,IPO_FRAME #BASE,POINT2[] " ",TQ_STATE FALSE}
DECL PDAT PPDAT79={ACC 100.000,APO_DIST 100.000,APO_MODE #CPTP,GEAR_JERK 50.0000}
DECL E6POS XP107={X 1293.96118,Y -629.543518,Z 1661.28882,A -62.0844460,B 76.3225,C 51.4223785,S 2,T 10,E1 190.873,E2 195.002197,E3 195.004211,E4 0.0,E5 0.0,E6 0.0}
DECL ATBg_Crater_T AC_WDAT59={JobModeId -187662529,ParamSetId -1375177600,CraterTime 0.100000,PostflowTime 0.100000,Channel1 30.0000,Channel2 1.00000,Channel3 0.0,Channel4 0.0,Channel5 0.0,Channel6 0.0,Channel7 0.0,Channel8 0.0,BurnBackTime 0.0}
DECL FDAT FP108={TOOL_NO 1,BASE_NO 0,IPO_FRAME #BASE,POINT2[] " ",TQ_STATE FALSE}
DECL LDAT LCPDAT32={ACC 100.000,APO_DIST 100.000,APO_FAC 50.0000,AXIS_VEL 100.000,AXIS_ACC 100.000,ORI_TYP #VAR,CIRC_TYP #BASE,JERK_FAC 50.0000,GEAR_JERK 50.0000,EXAX_IGN 0}
DECL E6POS XP108={X 1296.53784,Y -620.323242,Z 1661.69067,A -61.8037186,B 76.3528748,C 51.3231,S 2,T 10,E1 190.873,E2 195.002197,E3 195.004211,E4 0.0,E5 0.0,E6 0.0}
DECL ATBg_Start_T AS_WDAT60={JobModeId -187662529,ParamSetId 687014726,StartTime 0.0,PreFlowTime 0.100000,Channel1 30.0000,Channel2 1.00000,Channel3 0.0,Channel4 0.0,Channel5 0.0,Channel6 0.0,Channel7 0.0,Channel8 0.0,PurgeTime 0.0}
DECL ATBg_Weld_T AW_WDAT60={JobModeId -187662529,ParamSetId -430485013,Velocity 0.00830000,Channel1 30.0000,Channel2 1.00000,Channel3 0.0,Channel4 0.0,Channel5 0.0,Channel6 0.0,Channel7 0.0,Channel8 0.0}
DECL WTCg_WeaveDefinition_T WV_WDAT60={Pattern #None,Length 4.00000,Amplitude 2.00000,Angle 0.0}
DECL FDAT FP109={TOOL_NO 1,BASE_NO 0,IPO_FRAME #BASE,POINT2[] " ",TQ_STATE FALSE}
DECL PDAT PPDAT80={ACC 100.000,APO_DIST 100.000,APO_MODE #CPTP,GEAR_JERK 50.0000}
DECL E6POS XP109={X 1326.02588,Y -534.179382,Z 1641.57349,A -22.7906227,B 76.3941956,C 71.2853470,S 2,T 10,E1 190.872955,E2 195.002258,E3 195.004166,E4 0.0,E5 0.0,E6 0.0}
DECL ATBg_Crater_T AC_WDAT61={JobModeId -187662529,ParamSetId -1375177600,CraterTime 0.100000,PostflowTime 0.100000,Channel1 30.0000,Channel2 1.00000,Channel3 0.0,Channel4 0.0,Channel5 0.0,Channel6 0.0,Channel7 0.0,Channel8 0.0,BurnBackTime 0.0}
DECL FDAT FP110={TOOL_NO 1,BASE_NO 0,IPO_FRAME #BASE,POINT2[] " ",TQ_STATE FALSE}
DECL LDAT LCPDAT33={ACC 100.000,APO_DIST 100.000,APO_FAC 50.0000,AXIS_VEL 100.000,AXIS_ACC 100.000,ORI_TYP #VAR,CIRC_TYP #BASE,JERK_FAC 50.0000,GEAR_JERK 50.0000,EXAX_IGN 0}
DECL E6POS XP110={X 1323.19653,Y -542.751892,Z 1647.43872,A -43.1925316,B 73.3963852,C 51.5705795,S 2,T 10,E1 190.872955,E2 195.002258,E3 195.004166,E4 0.0,E5 0.0,E6 0.0}
DECL E6POS XP111={X 1280.34766,Y -555.961731,Z 1683.12561,A -42.7582092,B 71.8603516,C 53.2912,S 2,T 10,E1 190.872955,E2 195.002258,E3 195.004166,E4 0.0,E5 0.0,E6 0.0}
DECL FDAT FP111={TOOL_NO 1,BASE_NO 0,IPO_FRAME #BASE,POINT2[] " ",TQ_STATE FALSE}
DECL PDAT PPDAT81={VEL 100.000,ACC 100.000,APO_DIST 100.000,APO_MODE #CDIS,GEAR_JERK 50.0000,EXAX_IGN 3}
DECL E6POS XP112={X 1215.70911,Y -555.400269,Z 1739.47400,A -50.7764931,B 73.0435410,C 52.7764130,S 2,T 10,E1 190.872971,E2 195.002228,E3 195.004196,E4 0.0,E5 0.0,E6 0.0}
DECL FDAT FP112={TOOL_NO 1,BASE_NO 0,IPO_FRAME #BASE,POINT2[] " ",TQ_STATE FALSE}
DECL PDAT PPDAT82={VEL 100.000,ACC 100.000,APO_DIST 100.000,APO_MODE #CDIS,GEAR_JERK 50.0000,EXAX_IGN 3}
DECL ATBg_Start_T AS_WDAT62={JobModeId -187662529,ParamSetId 687014726,StartTime 0.0,PreFlowTime 0.100000,Channel1 30.0000,Channel2 1.00000,Channel3 0.0,Channel4 0.0,Channel5 0.0,Channel6 0.0,Channel7 0.0,Channel8 0.0,PurgeTime 0.0}
DECL ATBg_Weld_T AW_WDAT62={JobModeId -187662529,ParamSetId -430485013,Velocity 0.00830000,Channel1 30.0000,Channel2 1.00000,Channel3 0.0,Channel4 0.0,Channel5 0.0,Channel6 0.0,Channel7 0.0,Channel8 0.0}
DECL WTCg_WeaveDefinition_T WV_WDAT62={Pattern #None,Length 4.00000,Amplitude 2.00000,Angle 0.0}
DECL FDAT FP113={TOOL_NO 1,BASE_NO 0,IPO_FRAME #BASE,POINT2[] " ",TQ_STATE FALSE}
DECL PDAT PPDAT83={ACC 100.000,APO_DIST 100.000,APO_MODE #CPTP,GEAR_JERK 50.0000}
DECL E6POS XP113={X 1296.56372,Y -770.400757,Z 1543.47070,A 0.142972514,B -35.3954086,C -120.373474,S 0,T 34,E1 162.876816,E2 195.002243,E3 195.004135,E4 0.0,E5 0.0,E6 0.0}
DECL E6POS XP114={X 1032.96,Y -606.570557,Z 1836.64832,A 12.8797731,B -52.1382599,C -138.512726,S 0,T 38,E1 162.876816,E2 195.002243,E3 195.004135,E4 0.0,E5 0.0,E6 0.0}
DECL FDAT FP114={TOOL_NO 1,BASE_NO 0,IPO_FRAME #BASE,POINT2[] " ",TQ_STATE FALSE}
DECL PDAT PPDAT84={VEL 100.000,ACC 100.000,APO_DIST 100.000,APO_MODE #CDIS,GEAR_JERK 50.0000,EXAX_IGN 3}
DECL E6POS XP115={X 983.717468,Y -386.217621,Z 1912.19458,A 54.8041496,B -28.0464611,C -156.126465,S 0,T 42,E1 167.538651,E2 195.002243,E3 195.004135,E4 0.0,E5 0.0,E6 0.0}
DECL FDAT FP115={TOOL_NO 1,BASE_NO 0,IPO_FRAME #BASE,POINT2[] " ",TQ_STATE FALSE}
DECL PDAT PPDAT85={VEL 100.000,ACC 100.000,APO_DIST 100.000,APO_MODE #CDIS,GEAR_JERK 50.0000,EXAX_IGN 3}
DECL E6POS XP116={X 1127.12122,Y -538.175171,Z 1741.28772,A 86.2300110,B 45.5118370,C -178.934204,S 2,T 42,E1 180.834290,E2 195.002258,E3 195.004150,E4 0.0,E5 0.0,E6 0.0}
DECL FDAT FP116={TOOL_NO 1,BASE_NO 0,IPO_FRAME #BASE,POINT2[] " ",TQ_STATE FALSE}
DECL PDAT PPDAT86={VEL 100.000,ACC 100.000,APO_DIST 100.000,APO_MODE #CDIS,GEAR_JERK 50.0000,EXAX_IGN 3}
DECL E6POS XP117={X 1223.14966,Y -576.219177,Z 1689.56824,A 62.8018608,B 70.9648209,C 154.731369,S 2,T 10,E1 186.179565,E2 195.002258,E3 195.004166,E4 0.0,E5 0.0,E6 0.0}
DECL FDAT FP117={TOOL_NO 1,BASE_NO 0,IPO_FRAME #BASE,POINT2[] " ",TQ_STATE FALSE}
DECL PDAT PPDAT87={VEL 100.000,ACC 100.000,APO_DIST 100.000,APO_MODE #CDIS,GEAR_JERK 50.0000,EXAX_IGN 3}
DECL E6POS XP118={X 1019.43097,Y -480.945862,Z 1982.61938,A -73.3126068,B 40.0338173,C 23.4100742,S 2,T 10,E1 190.873,E2 195.002197,E3 195.004211,E4 0.0,E5 0.0,E6 0.0}
DECL FDAT FP118={TOOL_NO 1,BASE_NO 0,IPO_FRAME #BASE,POINT2[] " ",TQ_STATE FALSE}
DECL PDAT PPDAT88={VEL 100.000,ACC 100.000,APO_DIST 100.000,APO_MODE #CDIS,GEAR_JERK 50.0000,EXAX_IGN 3}
DECL E6POS XP119={X 1185.85767,Y -519.089905,Z 1836.84534,A -82.4992828,B 53.5618,C 21.6134605,S 2,T 10,E1 190.873,E2 195.002197,E3 195.004211,E4 0.0,E5 0.0,E6 0.0}
DECL FDAT FP119={TOOL_NO 1,BASE_NO 0,IPO_FRAME #BASE,POINT2[] " ",TQ_STATE FALSE}
DECL PDAT PPDAT89={VEL 100.000,ACC 100.000,APO_DIST 100.000,APO_MODE #CDIS,GEAR_JERK 50.0000,EXAX_IGN 3}
DECL ATBg_Crater_T AC_WDAT63={JobModeId -187662529,ParamSetId -1375177600,CraterTime 0.100000,PostflowTime 0.100000,Channel1 30.0000,Channel2 1.00000,Channel3 0.0,Channel4 0.0,Channel5 0.0,Channel6 0.0,Channel7 0.0,Channel8 0.0,BurnBackTime 0.0}
DECL FDAT FP120={TOOL_NO 1,BASE_NO 0,IPO_FRAME #BASE,POINT2[] " ",TQ_STATE FALSE}
DECL LDAT LCPDAT34={ACC 100.000,APO_DIST 100.000,APO_FAC 50.0000,AXIS_VEL 100.000,AXIS_ACC 100.000,ORI_TYP #VAR,CIRC_TYP #BASE,JERK_FAC 50.0000,GEAR_JERK 50.0000,EXAX_IGN 0}
DECL E6POS XP120={X 1296.40698,Y -769.839050,Z 1543.91675,A 0.220987946,B -35.3882370,C -120.418251,S 0,T 34,E1 162.887863,E2 195.002243,E3 195.004135,E4 0.0,E5 0.0,E6 0.0}
DECL E6POS XP121={X 1015.08203,Y -595.076965,Z 1861.00537,A 9.26292515,B -48.8289833,C -133.777206,S 0,T 38,E1 162.887863,E2 195.002243,E3 195.004135,E4 0.0,E5 0.0,E6 0.0}
DECL FDAT FP121={TOOL_NO 1,BASE_NO 0,IPO_FRAME #BASE,POINT2[] " ",TQ_STATE FALSE}
DECL PDAT PPDAT90={VEL 100.000,ACC 100.000,APO_DIST 100.000,APO_MODE #CDIS,GEAR_JERK 50.0000,EXAX_IGN 3}
DECL ATBg_Start_T AS_WDAT64={JobModeId -187662529,ParamSetId 687014726,StartTime 0.0,PreFlowTime 0.100000,Channel1 30.0000,Channel2 1.00000,Channel3 0.0,Channel4 0.0,Channel5 0.0,Channel6 0.0,Channel7 0.0,Channel8 0.0,PurgeTime 0.0}
DECL ATBg_Weld_T AW_WDAT64={JobModeId -187662529,ParamSetId -430485013,Velocity 0.00830000,Channel1 30.0000,Channel2 1.00000,Channel3 0.0,Channel4 0.0,Channel5 0.0,Channel6 0.0,Channel7 0.0,Channel8 0.0}
DECL WTCg_WeaveDefinition_T WV_WDAT64={Pattern #None,Length 4.00000,Amplitude 2.00000,Angle 0.0}
DECL FDAT FP122={TOOL_NO 1,BASE_NO 0,IPO_FRAME #BASE,POINT2[] " ",TQ_STATE FALSE}
DECL PDAT PPDAT91={ACC 100.000,APO_DIST 100.000,APO_MODE #CPTP,GEAR_JERK 50.0000}
DECL E6POS XP122={X 1467.58130,Y -240.404205,Z 1528.18201,A -1.93412697,B -32.3756,C -98.3877335,S 2,T 34,E1 162.887863,E2 195.002243,E3 195.004135,E4 0.0,E5 0.0,E6 0.0}
DECL ATBg_Crater_T AC_WDAT65={JobModeId -187662529,ParamSetId -1375177600,CraterTime 0.100000,PostflowTime 0.100000,Channel1 30.0000,Channel2 1.00000,Channel3 0.0,Channel4 0.0,Channel5 0.0,Channel6 0.0,Channel7 0.0,Channel8 0.0,BurnBackTime 0.0}
DECL FDAT FP123={TOOL_NO 1,BASE_NO 0,IPO_FRAME #BASE,POINT2[] " ",TQ_STATE FALSE}
DECL LDAT LCPDAT35={ACC 100.000,APO_DIST 100.000,APO_FAC 50.0000,AXIS_VEL 100.000,AXIS_ACC 100.000,ORI_TYP #VAR,CIRC_TYP #BASE,JERK_FAC 50.0000,GEAR_JERK 50.0000,EXAX_IGN 0}
DECL E6POS XP123={X 1467.58130,Y -240.404205,Z 1528.18201,A -1.93412697,B -32.3756,C -98.3877335,S 2,T 34,E1 162.887863,E2 195.002243,E3 195.004135,E4 0.0,E5 0.0,E6 0.0}
DECL ATBg_Start_T AS_WDAT66={JobModeId -187662529,ParamSetId 687014726,StartTime 0.0,PreFlowTime 0.100000,Channel1 30.0000,Channel2 1.00000,Channel3 0.0,Channel4 0.0,Channel5 0.0,Channel6 0.0,Channel7 0.0,Channel8 0.0,PurgeTime 0.0}
DECL ATBg_Weld_T AW_WDAT66={JobModeId -187662529,ParamSetId -430485013,Velocity 0.00830000,Channel1 30.0000,Channel2 1.00000,Channel3 0.0,Channel4 0.0,Channel5 0.0,Channel6 0.0,Channel7 0.0,Channel8 0.0}
DECL WTCg_WeaveDefinition_T WV_WDAT66={Pattern #None,Length 4.00000,Amplitude 2.00000,Angle 0.0}
DECL FDAT FP124={TOOL_NO 1,BASE_NO 0,IPO_FRAME #BASE,POINT2[] " ",TQ_STATE FALSE}
DECL PDAT PPDAT92={ACC 100.000,APO_DIST 100.000,APO_MODE #CPTP,GEAR_JERK 50.0000}
DECL E6POS XP124={X 1481.05737,Y 10.8651133,Z 1536.92859,A -3.71409750,B -32.3918381,C -85.6522675,S 2,T 42,E1 162.887863,E2 195.002243,E3 195.004135,E4 0.0,E5 0.0,E6 0.0}
DECL ATBg_Crater_T AC_WDAT67={JobModeId -187662529,ParamSetId -1375177600,CraterTime 0.100000,PostflowTime 0.100000,Channel1 30.0000,Channel2 1.00000,Channel3 0.0,Channel4 0.0,Channel5 0.0,Channel6 0.0,Channel7 0.0,Channel8 0.0,BurnBackTime 0.0}
DECL FDAT FP125={TOOL_NO 1,BASE_NO 0,IPO_FRAME #BASE,POINT2[] " ",TQ_STATE FALSE}
DECL LDAT LCPDAT36={ACC 100.000,APO_DIST 100.000,APO_FAC 50.0000,AXIS_VEL 100.000,AXIS_ACC 100.000,ORI_TYP #VAR,CIRC_TYP #BASE,JERK_FAC 50.0000,GEAR_JERK 50.0000,EXAX_IGN 0}
DECL E6POS XP125={X 1481.05737,Y 10.8651133,Z 1536.92859,A -3.71409750,B -32.3918381,C -85.6522675,S 2,T 42,E1 162.887863,E2 195.002243,E3 195.004135,E4 0.0,E5 0.0,E6 0.0}
DECL ATBg_Start_T AS_WDAT68={JobModeId -187662529,ParamSetId 687014726,StartTime 0.0,PreFlowTime 0.100000,Channel1 30.0000,Channel2 1.00000,Channel3 0.0,Channel4 0.0,Channel5 0.0,Channel6 0.0,Channel7 0.0,Channel8 0.0,PurgeTime 0.0}
DECL ATBg_Weld_T AW_WDAT68={JobModeId -187662529,ParamSetId -430485013,Velocity 0.00830000,Channel1 30.0000,Channel2 1.00000,Channel3 0.0,Channel4 0.0,Channel5 0.0,Channel6 0.0,Channel7 0.0,Channel8 0.0}
DECL WTCg_WeaveDefinition_T WV_WDAT68={Pattern #None,Length 4.00000,Amplitude 2.00000,Angle 0.0}
DECL FDAT FP126={TOOL_NO 1,BASE_NO 0,IPO_FRAME #BASE,POINT2[] " ",TQ_STATE FALSE}
DECL PDAT PPDAT93={ACC 100.000,APO_DIST 100.000,APO_MODE #CPTP,GEAR_JERK 50.0000}
DECL E6POS XP126={X 1444.21252,Y 329.091553,Z 1578.60730,A -4.10677433,B -37.4463387,C -75.4550400,S 2,T 43,E1 162.887848,E2 195.002243,E3 195.004120,E4 0.0,E5 0.0,E6 0.0}
DECL ATBg_Crater_T AC_WDAT69={JobModeId -187662529,ParamSetId -1375177600,CraterTime 0.100000,PostflowTime 0.100000,Channel1 30.0000,Channel2 1.00000,Channel3 0.0,Channel4 0.0,Channel5 0.0,Channel6 0.0,Channel7 0.0,Channel8 0.0,BurnBackTime 0.0}
DECL FDAT FP127={TOOL_NO 1,BASE_NO 0,IPO_FRAME #BASE,POINT2[] " ",TQ_STATE FALSE}
DECL LDAT LCPDAT37={ACC 100.000,APO_DIST 100.000,APO_FAC 50.0000,AXIS_VEL 100.000,AXIS_ACC 100.000,ORI_TYP #VAR,CIRC_TYP #BASE,JERK_FAC 50.0000,GEAR_JERK 50.0000,EXAX_IGN 0}
DECL E6POS XP127={X 1444.21252,Y 329.091553,Z 1578.60730,A -4.10677433,B -37.4463387,C -75.4550400,S 2,T 43,E1 162.887848,E2 195.002243,E3 195.004120,E4 0.0,E5 0.0,E6 0.0}
DECL ATBg_Start_T AS_WDAT70={JobModeId -187662529,ParamSetId 687014726,StartTime 0.0,PreFlowTime 0.100000,Channel1 30.0000,Channel2 1.00000,Channel3 0.0,Channel4 0.0,Channel5 0.0,Channel6 0.0,Channel7 0.0,Channel8 0.0,PurgeTime 0.0}
DECL ATBg_Weld_T AW_WDAT70={JobModeId -187662529,ParamSetId -430485013,Velocity 0.00830000,Channel1 30.0000,Channel2 1.00000,Channel3 0.0,Channel4 0.0,Channel5 0.0,Channel6 0.0,Channel7 0.0,Channel8 0.0}
DECL WTCg_WeaveDefinition_T WV_WDAT70={Pattern #None,Length 4.00000,Amplitude 2.00000,Angle 0.0}
DECL FDAT FP128={TOOL_NO 1,BASE_NO 0,IPO_FRAME #BASE,POINT2[] " ",TQ_STATE FALSE}
DECL PDAT PPDAT94={ACC 100.000,APO_DIST 100.000,APO_MODE #CPTP,GEAR_JERK 50.0000}
DECL E6POS XP128={X 1444.21252,Y 329.091553,Z 1578.60730,A -4.10677433,B -37.4463387,C -75.4550400,S 2,T 43,E1 162.887848,E2 195.002243,E3 195.004120,E4 0.0,E5 0.0,E6 0.0}
DECL ATBg_Crater_T AC_WDAT71={JobModeId -187662529,ParamSetId -1375177600,CraterTime 0.100000,PostflowTime 0.100000,Channel1 30.0000,Channel2 1.00000,Channel3 0.0,Channel4 0.0,Channel5 0.0,Channel6 0.0,Channel7 0.0,Channel8 0.0,BurnBackTime 0.0}
DECL FDAT FP129={TOOL_NO 1,BASE_NO 0,IPO_FRAME #BASE,POINT2[] " ",TQ_STATE FALSE}
DECL LDAT LCPDAT38={ACC 100.000,APO_DIST 100.000,APO_FAC 50.0000,AXIS_VEL 100.000,AXIS_ACC 100.000,ORI_TYP #VAR,CIRC_TYP #BASE,JERK_FAC 50.0000,GEAR_JERK 50.0000,EXAX_IGN 0}
DECL E6POS XP129={X 1444.21252,Y 329.091553,Z 1578.60730,A -4.10677433,B -37.4463387,C -75.4550400,S 2,T 43,E1 162.887848,E2 195.002243,E3 195.004120,E4 0.0,E5 0.0,E6 0.0}
DECL E6POS XP130={X 1106.52942,Y 227.610046,Z 1915.48096,A -12.1633968,B -55.2442207,C -66.5929108,S 2,T 43,E1 162.887848,E2 195.002243,E3 195.004120,E4 0.0,E5 0.0,E6 0.0}
DECL FDAT FP130={TOOL_NO 1,BASE_NO 0,IPO_FRAME #BASE,POINT2[] " ",TQ_STATE FALSE}
DECL PDAT PPDAT95={VEL 100.000,ACC 100.000,APO_DIST 100.000,APO_MODE #CDIS,GEAR_JERK 50.0000,EXAX_IGN 3}
DECL E6POS XP131={X 1047.66113,Y 425.531586,Z 1914.70532,A -17.3199234,B -49.3159409,C -53.3732643,S 2,T 43,E1 162.887848,E2 195.002243,E3 195.004120,E4 0.0,E5 0.0,E6 0.0}
DECL FDAT FP131={TOOL_NO 1,BASE_NO 0,IPO_FRAME #BASE,POINT2[] " ",TQ_STATE FALSE}
DECL PDAT PPDAT96={VEL 100.000,ACC 100.000,APO_DIST 100.000,APO_MODE #CDIS,GEAR_JERK 50.0000,EXAX_IGN 3}
DECL ATBg_Start_T AS_WDAT72={JobModeId -187662529,ParamSetId 687014726,StartTime 0.0,PreFlowTime 0.100000,Channel1 30.0000,Channel2 1.00000,Channel3 0.0,Channel4 0.0,Channel5 0.0,Channel6 0.0,Channel7 0.0,Channel8 0.0,PurgeTime 0.0}
DECL ATBg_Weld_T AW_WDAT72={JobModeId -187662529,ParamSetId -430485013,Velocity 0.00830000,Channel1 30.0000,Channel2 1.00000,Channel3 0.0,Channel4 0.0,Channel5 0.0,Channel6 0.0,Channel7 0.0,Channel8 0.0}
DECL WTCg_WeaveDefinition_T WV_WDAT72={Pattern #None,Length 4.00000,Amplitude 2.00000,Angle 0.0}
DECL FDAT FP132={TOOL_NO 1,BASE_NO 0,IPO_FRAME #BASE,POINT2[] " ",TQ_STATE FALSE}
DECL PDAT PPDAT97={ACC 100.000,APO_DIST 100.000,APO_MODE #CPTP,GEAR_JERK 50.0000}
DECL E6POS XP132={X 1380.53210,Y 589.161865,Z 1585.12817,A -0.785289049,B -38.0413094,C -68.7817764,S 2,T 43,E1 162.887848,E2 195.002243,E3 195.004120,E4 0.0,E5 0.0,E6 0.0}
DECL ATBg_Crater_T AC_WDAT73={JobModeId -187662529,ParamSetId -1375177600,CraterTime 0.100000,PostflowTime 0.100000,Channel1 30.0000,Channel2 1.00000,Channel3 0.0,Channel4 0.0,Channel5 0.0,Channel6 0.0,Channel7 0.0,Channel8 0.0,BurnBackTime 0.0}
DECL FDAT FP133={TOOL_NO 1,BASE_NO 0,IPO_FRAME #BASE,POINT2[] " ",TQ_STATE FALSE}
DECL LDAT LCPDAT39={ACC 100.000,APO_DIST 100.000,APO_FAC 50.0000,AXIS_VEL 100.000,AXIS_ACC 100.000,ORI_TYP #VAR,CIRC_TYP #BASE,JERK_FAC 50.0000,GEAR_JERK 50.0000,EXAX_IGN 0}
DECL E6POS XP133={X 1380.53210,Y 589.161865,Z 1585.12817,A -0.785289049,B -38.0413094,C -68.7817764,S 2,T 43,E1 162.887848,E2 195.002243,E3 195.004120,E4 0.0,E5 0.0,E6 0.0}
DECL ATBg_Start_T AS_WDAT74={JobModeId -187662529,ParamSetId 687014726,StartTime 0.0,PreFlowTime 0.100000,Channel1 30.0000,Channel2 1.00000,Channel3 0.0,Channel4 0.0,Channel5 0.0,Channel6 0.0,Channel7 0.0,Channel8 0.0,PurgeTime 0.0}
DECL ATBg_Weld_T AW_WDAT74={JobModeId -187662529,ParamSetId -430485013,Velocity 0.00830000,Channel1 30.0000,Channel2 1.00000,Channel3 0.0,Channel4 0.0,Channel5 0.0,Channel6 0.0,Channel7 0.0,Channel8 0.0}
DECL WTCg_WeaveDefinition_T WV_WDAT74={Pattern #None,Length 4.00000,Amplitude 2.00000,Angle 0.0}
DECL FDAT FP134={TOOL_NO 1,BASE_NO 0,IPO_FRAME #BASE,POINT2[] " ",TQ_STATE FALSE}
DECL PDAT PPDAT98={ACC 100.000,APO_DIST 100.000,APO_MODE #CPTP,GEAR_JERK 50.0000}
DECL E6POS XP134={X 1324.21606,Y 577.033569,Z 1675.84180,A 33.2802849,B 68.3659897,C 98.0990524,S 2,T 43,E1 193.523224,E2 195.002243,E3 195.004120,E4 0.0,E5 0.0,E6 0.0}
DECL ATBg_Crater_T AC_WDAT75={JobModeId -187662529,ParamSetId -1375177600,CraterTime 0.100000,PostflowTime 0.100000,Channel1 30.0000,Channel2 1.00000,Channel3 0.0,Channel4 0.0,Channel5 0.0,Channel6 0.0,Channel7 0.0,Channel8 0.0,BurnBackTime 0.0}
DECL FDAT FP135={TOOL_NO 1,BASE_NO 0,IPO_FRAME #BASE,POINT2[] " ",TQ_STATE FALSE}
DECL LDAT LCPDAT40={ACC 100.000,APO_DIST 100.000,APO_FAC 50.0000,AXIS_VEL 100.000,AXIS_ACC 100.000,ORI_TYP #VAR,CIRC_TYP #BASE,JERK_FAC 50.0000,GEAR_JERK 50.0000,EXAX_IGN 0}
DECL E6POS XP135={X 1315.22058,Y 580.528381,Z 1674.43982,A 33.6923904,B 68.7131882,C 98.2455063,S 2,T 43,E1 193.523224,E2 195.002243,E3 195.004120,E4 0.0,E5 0.0,E6 0.0}
DECL E6POS XP136={X 877.952393,Y 378.009613,Z 2066.49194,A 29.4934158,B 46.4165955,C 93.3650665,S 2,T 43,E1 66.3312759,E2 195.002243,E3 195.004120,E4 0.0,E5 0.0,E6 0.0}
DECL FDAT FP136={TOOL_NO 1,BASE_NO 0,IPO_FRAME #BASE,POINT2[] " ",TQ_STATE FALSE}
DECL PDAT PPDAT99={VEL 100.000,ACC 100.000,APO_DIST 100.000,APO_MODE #CDIS,GEAR_JERK 50.0000,EXAX_IGN 3}
DECL E6POS XP137={X 930.186890,Y 401.235260,Z 2032.07666,A 29.6696663,B 48.8887520,C 93.6704865,S 2,T 43,E1 117.250534,E2 195.002243,E3 195.004120,E4 0.0,E5 0.0,E6 0.0}
DECL FDAT FP137={TOOL_NO 1,BASE_NO 0,IPO_FRAME #BASE,POINT2[] " ",TQ_STATE FALSE}
DECL PDAT PPDAT100={VEL 100.000,ACC 100.000,APO_DIST 100.000,APO_MODE #CDIS,GEAR_JERK 50.0000,EXAX_IGN 3}
DECL E6POS XP138={X 1118.40247,Y -137.306046,Z 1876.11963,A 29.1699791,B -44.9447441,C -129.111099,S 2,T 34,E1 162.887863,E2 195.002243,E3 195.004135,E4 0.0,E5 0.0,E6 0.0}
DECL FDAT FP138={TOOL_NO 1,BASE_NO 0,IPO_FRAME #BASE,POINT2[] " ",TQ_STATE FALSE}
DECL PDAT PPDAT101={VEL 100.000,ACC 100.000,APO_DIST 100.000,APO_MODE #CDIS,GEAR_JERK 50.0000,EXAX_IGN 3}
DECL E6POS XP139={X 1118.40247,Y -137.306061,Z 1876.11963,A 29.1699696,B -44.9447479,C -129.111099,S 2,T 34,E1 162.887863,E2 195.002243,E3 195.004135,E4 0.0,E5 0.0,E6 0.0}
DECL FDAT FP139={TOOL_NO 1,BASE_NO 0,IPO_FRAME #BASE,POINT2[] " ",TQ_STATE FALSE}
DECL PDAT PPDAT102={VEL 100.000,ACC 100.000,APO_DIST 100.000,APO_MODE #CDIS,GEAR_JERK 50.0000,EXAX_IGN 3}
DECL E6POS XP140={X 1130.15820,Y 68.0121,Z 1887.62683,A 1.93376851,B -54.0676651,C -97.8631592,S 2,T 35,E1 162.887863,E2 195.002243,E3 195.004135,E4 0.0,E5 0.0,E6 0.0}
DECL FDAT FP140={TOOL_NO 1,BASE_NO 0,IPO_FRAME #BASE,POINT2[] " ",TQ_STATE FALSE}
DECL PDAT PPDAT103={VEL 100.000,ACC 100.000,APO_DIST 100.000,APO_MODE #CDIS,GEAR_JERK 50.0000,EXAX_IGN 3}
DECL E6POS XP141={X 1438.32813,Y 17.7426624,Z 1580.02771,A -3.33024645,B -33.9155655,C -86.5758896,S 2,T 42,E1 162.887863,E2 195.002243,E3 195.004135,E4 0.0,E5 0.0,E6 0.0}
DECL FDAT FP141={TOOL_NO 1,BASE_NO 0,IPO_FRAME #BASE,POINT2[] " ",TQ_STATE FALSE}
DECL PDAT PPDAT104={VEL 100.000,ACC 100.000,APO_DIST 100.000,APO_MODE #CDIS,GEAR_JERK 50.0000,EXAX_IGN 3}
DECL E6POS XP142={X 1438.32813,Y 17.7426624,Z 1580.02771,A -3.33024645,B -33.9155655,C -86.5758896,S 2,T 42,E1 162.887863,E2 195.002243,E3 195.004135,E4 0.0,E5 0.0,E6 0.0}
DECL FDAT FP142={TOOL_NO 1,BASE_NO 0,IPO_FRAME #BASE,POINT2[] " ",TQ_STATE FALSE}
DECL PDAT PPDAT105={VEL 100.000,ACC 100.000,APO_DIST 100.000,APO_MODE #CDIS,GEAR_JERK 50.0000,EXAX_IGN 3}
DECL E6POS XP143={X 1343.19556,Y 573.995483,Z 1631.42358,A -1.42052090,B -39.8733025,C -67.7716,S 2,T 43,E1 162.887848,E2 195.002243,E3 195.004120,E4 0.0,E5 0.0,E6 0.0}
DECL FDAT FP143={TOOL_NO 1,BASE_NO 0,IPO_FRAME #BASE,POINT2[] " ",TQ_STATE FALSE}
DECL PDAT PPDAT106={VEL 100.000,ACC 100.000,APO_DIST 100.000,APO_MODE #CDIS,GEAR_JERK 50.0000,EXAX_IGN 3}
DECL E6POS XP144={X 1273.17053,Y 587.464966,Z 1698.79993,A 83.2784653,B 60.5438156,C 145.168457,S 2,T 43,E1 190.194763,E2 195.002243,E3 195.004120,E4 0.0,E5 0.0,E6 0.0}
DECL FDAT FP144={TOOL_NO 1,BASE_NO 0,IPO_FRAME #BASE,POINT2[] " ",TQ_STATE FALSE}
DECL PDAT PPDAT107={VEL 100.000,ACC 100.000,APO_DIST 100.000,APO_MODE #CDIS,GEAR_JERK 50.0000,EXAX_IGN 3}
DECL ATBg_Start_T AS_WDAT76={JobModeId -187662529,ParamSetId 687014726,StartTime 0.0,PreFlowTime 0.100000,Channel1 30.0000,Channel2 1.00000,Channel3 0.0,Channel4 0.0,Channel5 0.0,Channel6 0.0,Channel7 0.0,Channel8 0.0,PurgeTime 0.0}
DECL ATBg_Weld_T AW_WDAT76={JobModeId -187662529,ParamSetId -430485013,Velocity 0.00830000,Channel1 30.0000,Channel2 1.00000,Channel3 0.0,Channel4 0.0,Channel5 0.0,Channel6 0.0,Channel7 0.0,Channel8 0.0}
DECL WTCg_WeaveDefinition_T WV_WDAT76={Pattern #None,Length 4.00000,Amplitude 2.00000,Angle 0.0}
DECL FDAT FP145={TOOL_NO 1,BASE_NO 0,IPO_FRAME #BASE,POINT2[] " ",TQ_STATE FALSE}
DECL PDAT PPDAT108={ACC 100.000,APO_DIST 100.000,APO_MODE #CPTP,GEAR_JERK 50.0000}
DECL E6POS XP145={X 1350.38965,Y 500.946869,Z 1633.47791,A 59.2960243,B 60.0680428,C 137.259659,S 6,T 27,E1 51.7690620,E2 195.002243,E3 195.004120,E4 0.0,E5 0.0,E6 0.0}
DECL ATBg_Crater_T AC_WDAT77={JobModeId -187662529,ParamSetId -1375177600,CraterTime 0.100000,PostflowTime 0.100000,Channel1 30.0000,Channel2 1.00000,Channel3 0.0,Channel4 0.0,Channel5 0.0,Channel6 0.0,Channel7 0.0,Channel8 0.0,BurnBackTime 0.0}
DECL FDAT FP146={TOOL_NO 1,BASE_NO 0,IPO_FRAME #BASE,POINT2[] " ",TQ_STATE FALSE}
DECL LDAT LCPDAT41={ACC 100.000,APO_DIST 100.000,APO_FAC 50.0000,AXIS_VEL 100.000,AXIS_ACC 100.000,ORI_TYP #VAR,CIRC_TYP #BASE,JERK_FAC 50.0000,GEAR_JERK 50.0000,EXAX_IGN 0}
DECL E6POS XP146={X 1350.38965,Y 500.946869,Z 1633.47791,A 59.2960243,B 60.0680428,C 137.259659,S 6,T 27,E1 51.7690620,E2 195.002243,E3 195.004120,E4 0.0,E5 0.0,E6 0.0}
DECL ATBg_Start_T AS_WDAT78={JobModeId -187662529,ParamSetId 687014726,StartTime 0.0,PreFlowTime 0.100000,Channel1 30.0000,Channel2 1.00000,Channel3 0.0,Channel4 0.0,Channel5 0.0,Channel6 0.0,Channel7 0.0,Channel8 0.0,PurgeTime 0.0}
DECL ATBg_Weld_T AW_WDAT78={JobModeId -187662529,ParamSetId -430485013,Velocity 0.00830000,Channel1 30.0000,Channel2 1.00000,Channel3 0.0,Channel4 0.0,Channel5 0.0,Channel6 0.0,Channel7 0.0,Channel8 0.0}
DECL WTCg_WeaveDefinition_T WV_WDAT78={Pattern #None,Length 4.00000,Amplitude 2.00000,Angle 0.0}
DECL FDAT FP147={TOOL_NO 1,BASE_NO 0,IPO_FRAME #BASE,POINT2[] " ",TQ_STATE FALSE}
DECL PDAT PPDAT109={ACC 100.000,APO_DIST 100.000,APO_MODE #CPTP,GEAR_JERK 50.0000}
DECL E6POS XP147={X 1393.22815,Y 126.055344,Z 1638.28113,A 24.8248920,B 64.7499,C 108.646500,S 6,T 27,E1 63.8692,E2 195.002243,E3 195.004120,E4 0.0,E5 0.0,E6 0.0}
DECL ATBg_Start_T AS_WDAT79={JobModeId -187662529,ParamSetId 687014726,StartTime 0.0,PreFlowTime 0.100000,Channel1 30.0000,Channel2 1.00000,Channel3 0.0,Channel4 0.0,Channel5 0.0,Channel6 0.0,Channel7 0.0,Channel8 0.0,PurgeTime 0.0}
DECL ATBg_Weld_T AW_WDAT79={JobModeId -187662529,ParamSetId -430485013,Velocity 0.00830000,Channel1 30.0000,Channel2 1.00000,Channel3 0.0,Channel4 0.0,Channel5 0.0,Channel6 0.0,Channel7 0.0,Channel8 0.0}
DECL WTCg_WeaveDefinition_T WV_WDAT79={Pattern #None,Length 4.00000,Amplitude 2.00000,Angle 0.0}
DECL FDAT FP148={TOOL_NO 1,BASE_NO 0,IPO_FRAME #BASE,POINT2[] " ",TQ_STATE FALSE}
DECL PDAT PPDAT110={ACC 100.000,APO_DIST 100.000,APO_MODE #CPTP,GEAR_JERK 50.0000}
DECL E6POS XP148={X 1391.42883,Y -96.0819855,Z 1637.99084,A 5.40315723,B 62.9757881,C 99.4957809,S 6,T 26,E1 63.8692,E2 195.002243,E3 195.004120,E4 0.0,E5 0.0,E6 0.0}
DECL ATBg_Crater_T AC_WDAT80={JobModeId -187662529,ParamSetId -1375177600,CraterTime 0.100000,PostflowTime 0.100000,Channel1 30.0000,Channel2 1.00000,Channel3 0.0,Channel4 0.0,Channel5 0.0,Channel6 0.0,Channel7 0.0,Channel8 0.0,BurnBackTime 0.0}
DECL FDAT FP149={TOOL_NO 1,BASE_NO 0,IPO_FRAME #BASE,POINT2[] " ",TQ_STATE FALSE}
DECL LDAT LCPDAT42={ACC 100.000,APO_DIST 100.000,APO_FAC 50.0000,AXIS_VEL 100.000,AXIS_ACC 100.000,ORI_TYP #VAR,CIRC_TYP #BASE,JERK_FAC 50.0000,GEAR_JERK 50.0000,EXAX_IGN 0}
DECL E6POS XP149={X 1391.42883,Y -96.0819855,Z 1637.99084,A 5.40315723,B 62.9757881,C 99.4957809,S 6,T 26,E1 63.8692,E2 195.002243,E3 195.004120,E4 0.0,E5 0.0,E6 0.0}
DECL ATBg_Start_T AS_WDAT81={JobModeId -187662529,ParamSetId 687014726,StartTime 0.0,PreFlowTime 0.100000,Channel1 30.0000,Channel2 1.00000,Channel3 0.0,Channel4 0.0,Channel5 0.0,Channel6 0.0,Channel7 0.0,Channel8 0.0,PurgeTime 0.0}
DECL ATBg_Weld_T AW_WDAT81={JobModeId -187662529,ParamSetId -430485013,Velocity 0.00830000,Channel1 30.0000,Channel2 1.00000,Channel3 0.0,Channel4 0.0,Channel5 0.0,Channel6 0.0,Channel7 0.0,Channel8 0.0}
DECL WTCg_WeaveDefinition_T WV_WDAT81={Pattern #None,Length 4.00000,Amplitude 2.00000,Angle 0.0}
DECL FDAT FP150={TOOL_NO 1,BASE_NO 0,IPO_FRAME #BASE,POINT2[] " ",TQ_STATE FALSE}
DECL PDAT PPDAT111={ACC 100.000,APO_DIST 100.000,APO_MODE #CPTP,GEAR_JERK 50.0000}
DECL E6POS XP150={X 1391.42883,Y -96.0819855,Z 1637.99084,A 5.40315723,B 62.9757881,C 99.4957809,S 6,T 26,E1 63.8692,E2 195.002243,E3 195.004120,E4 0.0,E5 0.0,E6 0.0}
DECL ATBg_Crater_T AC_WDAT82={JobModeId -187662529,ParamSetId -1375177600,CraterTime 0.100000,PostflowTime 0.100000,Channel1 30.0000,Channel2 1.00000,Channel3 0.0,Channel4 0.0,Channel5 0.0,Channel6 0.0,Channel7 0.0,Channel8 0.0,BurnBackTime 0.0}
DECL FDAT FP151={TOOL_NO 1,BASE_NO 0,IPO_FRAME #BASE,POINT2[] " ",TQ_STATE FALSE}
DECL LDAT LCPDAT43={ACC 100.000,APO_DIST 100.000,APO_FAC 50.0000,AXIS_VEL 100.000,AXIS_ACC 100.000,ORI_TYP #VAR,CIRC_TYP #BASE,JERK_FAC 50.0000,GEAR_JERK 50.0000,EXAX_IGN 0}
DECL E6POS XP151={X 1391.42883,Y -96.0819855,Z 1637.99084,A 5.40315723,B 62.9757881,C 99.4957809,S 6,T 26,E1 63.8692,E2 195.002243,E3 195.004120,E4 0.0,E5 0.0,E6 0.0}
DECL ATBg_Start_T AS_WDAT83={JobModeId -187662529,ParamSetId 687014726,StartTime 0.0,PreFlowTime 0.100000,Channel1 30.0000,Channel2 1.00000,Channel3 0.0,Channel4 0.0,Channel5 0.0,Channel6 0.0,Channel7 0.0,Channel8 0.0,PurgeTime 0.0}
DECL ATBg_Weld_T AW_WDAT83={JobModeId -187662529,ParamSetId -430485013,Velocity 0.00830000,Channel1 30.0000,Channel2 1.00000,Channel3 0.0,Channel4 0.0,Channel5 0.0,Channel6 0.0,Channel7 0.0,Channel8 0.0}
DECL WTCg_WeaveDefinition_T WV_WDAT83={Pattern #None,Length 4.00000,Amplitude 2.00000,Angle 0.0}
DECL FDAT FP152={TOOL_NO 1,BASE_NO 0,IPO_FRAME #BASE,POINT2[] " ",TQ_STATE FALSE}
DECL PDAT PPDAT112={ACC 100.000,APO_DIST 100.000,APO_MODE #CPTP,GEAR_JERK 50.0000}
DECL E6POS XP152={X 1338.18860,Y -536.074524,Z 1647.32874,A -57.8892822,B 63.7091942,C 41.0981369,S 2,T 10,E1 63.8692,E2 195.002243,E3 195.004120,E4 0.0,E5 0.0,E6 0.0}
DECL ATBg_Crater_T AC_WDAT84={JobModeId -187662529,ParamSetId -1375177600,CraterTime 0.100000,PostflowTime 0.100000,Channel1 30.0000,Channel2 1.00000,Channel3 0.0,Channel4 0.0,Channel5 0.0,Channel6 0.0,Channel7 0.0,Channel8 0.0,BurnBackTime 0.0}
DECL FDAT FP153={TOOL_NO 1,BASE_NO 0,IPO_FRAME #BASE,POINT2[] " ",TQ_STATE FALSE}
DECL LDAT LCPDAT44={ACC 100.000,APO_DIST 100.000,APO_FAC 50.0000,AXIS_VEL 100.000,AXIS_ACC 100.000,ORI_TYP #VAR,CIRC_TYP #BASE,JERK_FAC 50.0000,GEAR_JERK 50.0000,EXAX_IGN 0}
DECL E6POS XP153={X 1338.18860,Y -536.074524,Z 1647.32874,A -57.8892822,B 63.7091942,C 41.0981369,S 2,T 10,E1 63.8692,E2 195.002243,E3 195.004120,E4 0.0,E5 0.0,E6 0.0}
DECL ATBg_Start_T AS_WDAT85={JobModeId -187662529,ParamSetId 687014726,StartTime 0.0,PreFlowTime 0.100000,Channel1 30.0000,Channel2 1.00000,Channel3 0.0,Channel4 0.0,Channel5 0.0,Channel6 0.0,Channel7 0.0,Channel8 0.0,PurgeTime 0.0}
DECL ATBg_Weld_T AW_WDAT85={JobModeId -187662529,ParamSetId -430485013,Velocity 0.00830000,Channel1 30.0000,Channel2 1.00000,Channel3 0.0,Channel4 0.0,Channel5 0.0,Channel6 0.0,Channel7 0.0,Channel8 0.0}
DECL WTCg_WeaveDefinition_T WV_WDAT85={Pattern #None,Length 4.00000,Amplitude 2.00000,Angle 0.0}
DECL FDAT FP154={TOOL_NO 1,BASE_NO 0,IPO_FRAME #BASE,POINT2[] " ",TQ_STATE FALSE}
DECL PDAT PPDAT113={ACC 100.000,APO_DIST 100.000,APO_MODE #CPTP,GEAR_JERK 50.0000}
DECL E6POS XP154={X 1262.58118,Y -864.338440,Z 1614.00354,A -73.6334381,B 51.8891182,C 20.1776752,S 2,T 10,E1 63.8692,E2 195.002243,E3 195.004120,E4 0.0,E5 0.0,E6 0.0}
DECL ATBg_Crater_T AC_WDAT86={JobModeId -187662529,ParamSetId -1375177600,CraterTime 0.100000,PostflowTime 0.100000,Channel1 30.0000,Channel2 1.00000,Channel3 0.0,Channel4 0.0,Channel5 0.0,Channel6 0.0,Channel7 0.0,Channel8 0.0,BurnBackTime 0.0}
DECL FDAT FP155={TOOL_NO 1,BASE_NO 0,IPO_FRAME #BASE,POINT2[] " ",TQ_STATE FALSE}
DECL LDAT LCPDAT45={ACC 100.000,APO_DIST 100.000,APO_FAC 50.0000,AXIS_VEL 100.000,AXIS_ACC 100.000,ORI_TYP #VAR,CIRC_TYP #BASE,JERK_FAC 50.0000,GEAR_JERK 50.0000,EXAX_IGN 0}
DECL E6POS XP155={X 1262.58118,Y -864.338440,Z 1614.00354,A -73.6334381,B 51.8891182,C 20.1776752,S 2,T 10,E1 63.8692,E2 195.002243,E3 195.004120,E4 0.0,E5 0.0,E6 0.0}
DECL E6POS XP156={X 1161.57153,Y -787.106750,Z 1730.94080,A -70.7340851,B 48.4049530,C 23.9520893,S 2,T 10,E1 63.8692,E2 195.002243,E3 195.004120,E4 0.0,E5 0.0,E6 0.0}
DECL FDAT FP156={TOOL_NO 1,BASE_NO 0,IPO_FRAME #BASE,POINT2[] " ",TQ_STATE FALSE}
DECL PDAT PPDAT114={VEL 100.000,ACC 100.000,APO_DIST 100.000,APO_MODE #CDIS,GEAR_JERK 50.0000,EXAX_IGN 3}
DECL E6POS XP157={X 1126.74866,Y 408.069397,Z 1841.40271,A 51.3672,B 51.7329292,C 127.716705,S 6,T 27,E1 51.7690620,E2 195.002243,E3 195.004120,E4 0.0,E5 0.0,E6 0.0}
DECL FDAT FP157={TOOL_NO 1,BASE_NO 0,IPO_FRAME #BASE,POINT2[] " ",TQ_STATE FALSE}
DECL PDAT PPDAT115={VEL 100.000,ACC 100.000,APO_DIST 100.000,APO_MODE #CDIS,GEAR_JERK 50.0000,EXAX_IGN 3}
DECL E6POS XP158={X 1302.66907,Y 210.702881,Z 1692.58154,A 8.67756748,B 64.1599197,C 93.2300949,S 6,T 27,E1 59.8376503,E2 195.002243,E3 195.004120,E4 0.0,E5 0.0,E6 0.0}
DECL FDAT FP158={TOOL_NO 1,BASE_NO 0,IPO_FRAME #BASE,POINT2[] " ",TQ_STATE FALSE}
DECL PDAT PPDAT116={VEL 100.000,ACC 100.000,APO_DIST 100.000,APO_MODE #CDIS,GEAR_JERK 50.0000,EXAX_IGN 3}
DECL E6POS XP159={X 1321.23755,Y 118.253990,Z 1679.97705,A 23.9074345,B 63.3932915,C 107.626610,S 6,T 27,E1 63.8688583,E2 195.002243,E3 195.004120,E4 0.0,E5 0.0,E6 0.0}
DECL FDAT FP159={TOOL_NO 1,BASE_NO 0,IPO_FRAME #BASE,POINT2[] " ",TQ_STATE FALSE}
DECL PDAT PPDAT117={VEL 100.000,ACC 100.000,APO_DIST 100.000,APO_MODE #CDIS,GEAR_JERK 50.0000,EXAX_IGN 3}
DECL ATBg_Crater_T AC_WDAT87={JobModeId -187662529,ParamSetId -1375177600,CraterTime 0.100000,PostflowTime 0.100000,Channel1 30.0000,Channel2 1.00000,Channel3 0.0,Channel4 0.0,Channel5 0.0,Channel6 0.0,Channel7 0.0,Channel8 0.0,BurnBackTime 0.0}
DECL FDAT FP160={TOOL_NO 1,BASE_NO 0,IPO_FRAME #BASE,POINT2[] " ",TQ_STATE FALSE}
DECL LDAT LCPDAT46={ACC 100.000,APO_DIST 100.000,APO_FAC 50.0000,AXIS_VEL 100.000,AXIS_ACC 100.000,ORI_TYP #VAR,CIRC_TYP #BASE,JERK_FAC 50.0000,GEAR_JERK 50.0000,EXAX_IGN 0}
DECL E6POS XP160={X 1393.22815,Y 126.055344,Z 1638.28113,A 24.8248920,B 64.7499,C 108.646500,S 6,T 27,E1 63.8692,E2 195.002243,E3 195.004120,E4 0.0,E5 0.0,E6 0.0}
DECL E6POS XP161={X 1172.91736,Y 102.155952,Z 1791.00903,A 21.1160088,B 58.0485039,C 104.429794,S 6,T 27,E1 63.8692,E2 195.002243,E3 195.004120,E4 0.0,E5 0.0,E6 0.0}
DECL FDAT FP161={TOOL_NO 1,BASE_NO 0,IPO_FRAME #BASE,POINT2[] " ",TQ_STATE FALSE}
DECL PDAT PPDAT118={VEL 100.000,ACC 100.000,APO_DIST 100.000,APO_MODE #CDIS,GEAR_JERK 50.0000,EXAX_IGN 3}
DECL E6POS XP162={X 1319.45740,Y -94.4541702,Z 1687.76807,A 6.00046062,B 61.2865181,C 99.9257813,S 6,T 26,E1 63.8692,E2 195.002243,E3 195.004120,E4 0.0,E5 0.0,E6 0.0}
DECL FDAT FP162={TOOL_NO 1,BASE_NO 0,IPO_FRAME #BASE,POINT2[] " ",TQ_STATE FALSE}
DECL PDAT PPDAT119={VEL 100.000,ACC 100.000,APO_DIST 100.000,APO_MODE #CDIS,GEAR_JERK 50.0000,EXAX_IGN 3}
DECL E6POS XP163={X 1105.24890,Y -83.5208740,Z 1816.11963,A 3.68451500,B 54.5741844,C 97.4914474,S 6,T 26,E1 63.8692,E2 195.002243,E3 195.004120,E4 0.0,E5 0.0,E6 0.0}
DECL FDAT FP163={TOOL_NO 1,BASE_NO 0,IPO_FRAME #BASE,POINT2[] " ",TQ_STATE FALSE}
DECL PDAT PPDAT120={VEL 100.000,ACC 100.000,APO_DIST 100.000,APO_MODE #CDIS,GEAR_JERK 50.0000,EXAX_IGN 3}
DECL E6POS XP164={X 1116.65540,Y -300.466644,Z 1807.37952,A -30.0061340,B 65.1442947,C 72.6307373,S 2,T 10,E1 63.8692,E2 195.002243,E3 195.004120,E4 0.0,E5 0.0,E6 0.0}
DECL FDAT FP164={TOOL_NO 1,BASE_NO 0,IPO_FRAME #BASE,POINT2[] " ",TQ_STATE FALSE}
DECL PDAT PPDAT121={VEL 100.000,ACC 100.000,APO_DIST 100.000,APO_MODE #CDIS,GEAR_JERK 50.0000,EXAX_IGN 3}
DECL E6POS XP165={X 1094.76465,Y -436.932404,Z 1850.25781,A -49.5495834,B 55.7893753,C 50.7237625,S 2,T 10,E1 63.8692,E2 195.002243,E3 195.004120,E4 0.0,E5 0.0,E6 0.0}
DECL FDAT FP165={TOOL_NO 1,BASE_NO 0,IPO_FRAME #BASE,POINT2[] " ",TQ_STATE FALSE}
DECL PDAT PPDAT122={VEL 100.000,ACC 100.000,APO_DIST 100.000,APO_MODE #CDIS,GEAR_JERK 50.0000,EXAX_IGN 3}
DECL E6POS XP166={X 1051.96350,Y -673.004822,Z 1817.49390,A -63.4329147,B 55.2390823,C 44.4735641,S 2,T 10,E1 63.8692,E2 195.002243,E3 195.004120,E4 0.0,E5 0.0,E6 0.0}
DECL FDAT FP166={TOOL_NO 1,BASE_NO 0,IPO_FRAME #BASE,POINT2[] " ",TQ_STATE FALSE}
DECL PDAT PPDAT123={VEL 100.000,ACC 100.000,APO_DIST 100.000,APO_MODE #CDIS,GEAR_JERK 50.0000,EXAX_IGN 3}
DECL ATBg_Start_T AS_WDAT88={JobModeId -187662529,ParamSetId 687014726,StartTime 0.0,PreFlowTime 0.100000,Channel1 30.0000,Channel2 1.00000,Channel3 0.0,Channel4 0.0,Channel5 0.0,Channel6 0.0,Channel7 0.0,Channel8 0.0,PurgeTime 0.0}
DECL ATBg_Weld_T AW_WDAT88={JobModeId -187662529,ParamSetId -430485013,Velocity 0.00830000,Channel1 30.0000,Channel2 1.00000,Channel3 0.0,Channel4 0.0,Channel5 0.0,Channel6 0.0,Channel7 0.0,Channel8 0.0}
DECL WTCg_WeaveDefinition_T WV_WDAT88={Pattern #None,Length 4.00000,Amplitude 2.00000,Angle 0.0}
DECL FDAT FP167={TOOL_NO 1,BASE_NO 0,IPO_FRAME #BASE,POINT2[] " ",TQ_STATE FALSE}
DECL PDAT PPDAT124={ACC 100.000,APO_DIST 100.000,APO_MODE #CPTP,GEAR_JERK 50.0000}
DECL E6POS XP167={X 1345.89380,Y -689.801575,Z 1567.35449,A 4.44710493,B -38.9034271,C -121.049332,S 0,T 34,E1 -15.0944824,E2 195.002243,E3 195.004120,E4 0.0,E5 0.0,E6 0.0}
DECL ATBg_Crater_T AC_WDAT89={JobModeId -187662529,ParamSetId -1375177600,CraterTime 0.100000,PostflowTime 0.100000,Channel1 30.0000,Channel2 1.00000,Channel3 0.0,Channel4 0.0,Channel5 0.0,Channel6 0.0,Channel7 0.0,Channel8 0.0,BurnBackTime 0.0}
DECL FDAT FP168={TOOL_NO 1,BASE_NO 0,IPO_FRAME #BASE,POINT2[] " ",TQ_STATE FALSE}
DECL LDAT LCPDAT47={ACC 100.000,APO_DIST 100.000,APO_FAC 50.0000,AXIS_VEL 100.000,AXIS_ACC 100.000,ORI_TYP #VAR,CIRC_TYP #BASE,JERK_FAC 50.0000,GEAR_JERK 50.0000,EXAX_IGN 0}
DECL E6POS XP168={X 1345.89380,Y -689.801575,Z 1567.35449,A 4.44710493,B -38.9034271,C -121.049332,S 0,T 34,E1 -15.0944824,E2 195.002243,E3 195.004120,E4 0.0,E5 0.0,E6 0.0}
DECL E6POS XP169={X 1115.44019,Y -564.918457,Z 1826.14063,A 11.2815619,B -48.6033707,C -130.884140,S 0,T 34,E1 -15.0944824,E2 195.002243,E3 195.004120,E4 0.0,E5 0.0,E6 0.0}
DECL FDAT FP169={TOOL_NO 1,BASE_NO 0,IPO_FRAME #BASE,POINT2[] " ",TQ_STATE FALSE}
DECL PDAT PPDAT125={VEL 100.000,ACC 100.000,APO_DIST 100.000,APO_MODE #CDIS,GEAR_JERK 50.0000,EXAX_IGN 3}
DECL ATBg_Start_T AS_WDAT90={JobModeId -187662529,ParamSetId 687014726,StartTime 0.0,PreFlowTime 0.100000,Channel1 30.0000,Channel2 1.00000,Channel3 0.0,Channel4 0.0,Channel5 0.0,Channel6 0.0,Channel7 0.0,Channel8 0.0,PurgeTime 0.0}
DECL ATBg_Weld_T AW_WDAT90={JobModeId -187662529,ParamSetId -430485013,Velocity 0.00830000,Channel1 30.0000,Channel2 1.00000,Channel3 0.0,Channel4 0.0,Channel5 0.0,Channel6 0.0,Channel7 0.0,Channel8 0.0}
DECL WTCg_WeaveDefinition_T WV_WDAT90={Pattern #None,Length 4.00000,Amplitude 2.00000,Angle 0.0}
DECL FDAT FP170={TOOL_NO 1,BASE_NO 0,IPO_FRAME #BASE,POINT2[] " ",TQ_STATE FALSE}
DECL PDAT PPDAT126={ACC 100.000,APO_DIST 100.000,APO_MODE #CPTP,GEAR_JERK 50.0000}
DECL E6POS XP170={X 1430.27856,Y -431.329437,Z 1568.64136,A -0.463984519,B -40.1669731,C -106.484306,S 2,T 34,E1 -15.0944824,E2 195.002243,E3 195.004120,E4 0.0,E5 0.0,E6 0.0}
DECL ATBg_Crater_T AC_WDAT91={JobModeId -187662529,ParamSetId -1375177600,CraterTime 0.100000,PostflowTime 0.100000,Channel1 30.0000,Channel2 1.00000,Channel3 0.0,Channel4 0.0,Channel5 0.0,Channel6 0.0,Channel7 0.0,Channel8 0.0,BurnBackTime 0.0}
DECL FDAT FP171={TOOL_NO 1,BASE_NO 0,IPO_FRAME #BASE,POINT2[] " ",TQ_STATE FALSE}
DECL LDAT LCPDAT48={ACC 100.000,APO_DIST 100.000,APO_FAC 50.0000,AXIS_VEL 100.000,AXIS_ACC 100.000,ORI_TYP #VAR,CIRC_TYP #BASE,JERK_FAC 50.0000,GEAR_JERK 50.0000,EXAX_IGN 0}
DECL E6POS XP171={X 1430.27856,Y -431.329437,Z 1568.64136,A -0.463984519,B -40.1669731,C -106.484306,S 2,T 34,E1 -15.0944824,E2 195.002243,E3 195.004120,E4 0.0,E5 0.0,E6 0.0}
